LIN {X 0,Y 370.499,Z 396.613,A -85,B 0,C 180,E1 -12676.286,E2 -12676.286} C_VEL
LIN {X 0,Y 370.097,Z 408.814,A -85,B 0,C 180,E1 -12676.83,E2 -12676.83} C_VEL
LIN {X 0,Y 369.553,Z 419.294,A -85,B 0,C 180,E1 -12677.509,E2 -12677.509} C_VEL
LIN {X 0,Y 369.157,Z 427.534,A -85,B 0,C 180,E1 -12678.193,E2 -12678.193} C_VEL
LIN {X 0,Y 368.756,Z 436.851,A -85,B 0,C 180,E1 -12679.154,E2 -12679.154} C_VEL
LIN {X 0,Y 368.3,Z 446.273,A -85,B 0,C 180,E1 -12680.39,E2 -12680.39} C_VEL
LIN {X 0,Y 368.015,Z 452.98,A -85,B 0,C 180,E1 -12681.491,E2 -12681.491} C_VEL
LIN {X 0,Y 367.806,Z 458.55,A -85,B 0,C 180,E1 -12682.591,E2 -12682.591} C_VEL
LIN {X 0,Y 367.616,Z 463.595,A -85,B 0,C 180,E1 -12683.807,E2 -12683.807} C_VEL
LIN {X 0,Y 367.587,Z 467.801,A -85,B 0,C 180,E1 -12685.066,E2 -12685.066} C_VEL
LIN {X 0,Y 367.464,Z 470.726,A -85,B 0,C 180,E1 -12686.164,E2 -12686.164} C_VEL
LIN {X 0,Y 367.501,Z 473.873,A -85,B 0,C 180,E1 -12687.81,E2 -12687.81} C_VEL
LIN {X 0,Y 367.55,Z 475.255,A -85,B 0,C 180,E1 -12688.906,E2 -12688.906} C_VEL
LIN {X 0,Y 367.528,Z 476.096,A -85,B 0,C 180,E1 -12690.002,E2 -12690.002} C_VEL
LIN {X 0,Y 367.446,Z 476.353,A -85,B 0,C 180,E1 -12691.098,E2 -12691.098} C_VEL
LIN {X 0,Y 367.379,Z 475.995,A -85,B 0,C 180,E1 -12692.195,E2 -12692.195} C_VEL
LIN {X 0,Y 367.4,Z 475.12,A -85,B 0,C 180,E1 -12693.292,E2 -12693.292} C_VEL
LIN {X 0,Y 367.518,Z 473.725,A -85,B 0,C 180,E1 -12694.389,E2 -12694.389} C_VEL
LIN {X 0,Y 367.552,Z 471.788,A -85,B 0,C 180,E1 -12695.488,E2 -12695.488} C_VEL
LIN {X 0,Y 367.703,Z 469.247,A -85,B 0,C 180,E1 -12696.587,E2 -12696.587} C_VEL
LIN {X 0,Y 368.146,Z 464.102,A -85,B 0,C 180,E1 -12698.233,E2 -12698.233} C_VEL
LIN {X 0,Y 368.658,Z 458.565,A -85,B 0,C 180,E1 -12699.604,E2 -12699.604} C_VEL
LIN {X 0,Y 369.267,Z 453.206,A -85,B 0,C 180,E1 -12700.696,E2 -12700.696} C_VEL
LIN {X 0,Y 369.939,Z 446.802,A -85,B 0,C 180,E1 -12701.786,E2 -12701.786} C_VEL
LIN {X 0,Y 370.677,Z 439.081,A -85,B 0,C 180,E1 -12702.874,E2 -12702.874} C_VEL
LIN {X 0,Y 371.679,Z 429.594,A -85,B 0,C 180,E1 -12703.952,E2 -12703.952} C_VEL
LIN {X 0,Y 372.685,Z 418.758,A -85,B 0,C 180,E1 -12704.89,E2 -12704.89} C_VEL
LIN {X 0,Y 373.447,Z 409.895,A -85,B 0,C 180,E1 -12705.487,E2 -12705.487} C_VEL
LIN {X 0,Y 374.208,Z 399.587,A -85,B 0,C 180,E1 -12706.014,E2 -12706.014} C_VEL
LIN {X 0,Y 374.95,Z 384.489,A -85,B 0,C 180,E1 -12706.523,E2 -12706.523} C_VEL
LIN {X 0,Y 376.379,Z 344.678,A -85,B 0,C 180,E1 -12707.661,E2 -12707.661} C_VEL
LIN {X 0,Y 374.795,Z 331.794,A -85,B 0,C 180,E1 -12708.21,E2 -12708.21} C_VEL
LIN {X 0,Y 371.759,Z 316.775,A -85,B 0,C 180,E1 -12708.987,E2 -12708.987} C_VEL
LIN {X 0,Y 370.823,Z 312.912,A -85,B 0,C 180,E1 -12709.212,E2 -12709.212} C_VEL
LIN {X 0,Y 371.941,Z 296.849,A -85,B 0,C 180,E1 -12712.792,E2 -12712.792} C_VEL
LIN {X 0,Y 372.152,Z 293.067,A -85,B 0,C 180,E1 -12713.661,E2 -12713.661} C_VEL
LIN {X 0,Y 370.264,Z 284.467,A -85,B 0,C 180,E1 -12715.887,E2 -12715.887} C_VEL
LIN {X 0,Y 368.901,Z 279.352,A -85,B 0,C 180,E1 -12717.287,E2 -12717.287} C_VEL
LIN {X 0,Y 368.905,Z 279.348,A -85,B 0,C 180,E1 -12720.981,E2 -12720.981} C_VEL
LIN {X 0,Y 368.887,Z 279.348,A -85,B 0,C 180,E1 -12724.987,E2 -12724.987} C_VEL
LIN {X 0,Y 368.888,Z 279.346,A -85,B 0,C 180,E1 -12728.632,E2 -12728.632} C_VEL
LIN {X 0,Y 368.871,Z 279.346,A -85,B 0,C 180,E1 -12732.003,E2 -12732.003} C_VEL
LIN {X 0,Y 368.866,Z 279.35,A -85,B 0,C 180,E1 -12735.169,E2 -12735.169} C_VEL
LIN {X 0,Y 368.874,Z 279.344,A -85,B 0,C 180,E1 -12738.172,E2 -12738.172} C_VEL
LIN {X 0,Y 368.894,Z 279.342,A -85,B 0,C 180,E1 -12741.364,E2 -12741.364} C_VEL
LIN {X 0,Y 368.949,Z 279.338,A -85,B 0,C 180,E1 -12745.143,E2 -12745.143} C_VEL
LIN {X 0,Y 368.931,Z 279.342,A -85,B 0,C 180,E1 -12749.042,E2 -12749.042} C_VEL
LIN {X 0,Y 368.93,Z 279.345,A -85,B 0,C 180,E1 -12751.555,E2 -12751.555} C_VEL
LIN {X 0,Y 368.943,Z 279.346,A -85,B 0,C 180,E1 -12755.219,E2 -12755.219} C_VEL
LIN {X 0,Y 368.959,Z 279.518,A -85,B 0,C 180,E1 -12758.558,E2 -12758.558} C_VEL
LIN {X 0,Y 372.025,Z 289.625,A -85,B 0,C 180,E1 -12760.867,E2 -12760.867} C_VEL
LIN {X 0,Y 375.275,Z 296.975,A -85,B 0,C 180,E1 -12761.431,E2 -12761.431} C_VEL
LIN {X 0,Y 377.46,Z 310.343,A -85,B 0,C 180,E1 -12762.076,E2 -12762.076} C_VEL
LIN {X 0,Y 374.942,Z 371.825,A -85,B 0,C 180,E1 -12763.875,E2 -12763.875} C_VEL
LIN {X 0,Y 374.226,Z 384.155,A -85,B 0,C 180,E1 -12764.473,E2 -12764.473} C_VEL
LIN {X 0,Y 373.553,Z 393.994,A -85,B 0,C 180,E1 -12765.142,E2 -12765.142} C_VEL
LIN {X 0,Y 372.837,Z 403.308,A -85,B 0,C 180,E1 -12765.95,E2 -12765.95} C_VEL
LIN {X 0,Y 371.896,Z 413.125,A -85,B 0,C 180,E1 -12767.027,E2 -12767.027} C_VEL
LIN {X 0,Y 371.065,Z 421.69,A -85,B 0,C 180,E1 -12768.247,E2 -12768.247} C_VEL
LIN {X 0,Y 370.327,Z 427.955,A -85,B 0,C 180,E1 -12769.332,E2 -12769.332} C_VEL
LIN {X 0,Y 369.723,Z 433.161,A -85,B 0,C 180,E1 -12770.421,E2 -12770.421} C_VEL
LIN {X 0,Y 369.172,Z 437.83,A -85,B 0,C 180,E1 -12771.606,E2 -12771.606} C_VEL
LIN {X 0,Y 368.614,Z 442.264,A -85,B 0,C 180,E1 -12773.019,E2 -12773.019} C_VEL
LIN {X 0,Y 368.055,Z 445.796,A -85,B 0,C 180,E1 -12774.516,E2 -12774.516} C_VEL
LIN {X 0,Y 368.038,Z 447.581,A -85,B 0,C 180,E1 -12775.614,E2 -12775.614} C_VEL
LIN {X 0,Y 367.844,Z 448.849,A -85,B 0,C 180,E1 -12776.709,E2 -12776.709} C_VEL
LIN {X 0,Y 367.656,Z 449.603,A -85,B 0,C 180,E1 -12777.804,E2 -12777.804} C_VEL
LIN {X 0,Y 367.542,Z 449.826,A -85,B 0,C 180,E1 -12778.899,E2 -12778.899} C_VEL
LIN {X 0,Y 367.511,Z 449.429,A -85,B 0,C 180,E1 -12779.994,E2 -12779.994} C_VEL
LIN {X 0,Y 367.468,Z 448.484,A -85,B 0,C 180,E1 -12781.09,E2 -12781.09} C_VEL
LIN {X 0,Y 367.501,Z 446.123,A -85,B 0,C 180,E1 -12782.735,E2 -12782.735} C_VEL
LIN {X 0,Y 367.672,Z 442.383,A -85,B 0,C 180,E1 -12784.379,E2 -12784.379} C_VEL
LIN {X 0,Y 367.762,Z 437.898,A -85,B 0,C 180,E1 -12785.805,E2 -12785.805} C_VEL
LIN {X 0,Y 368.03,Z 432.871,A -85,B 0,C 180,E1 -12787.069,E2 -12787.069} C_VEL
LIN {X 0,Y 368.285,Z 427.255,A -85,B 0,C 180,E1 -12788.223,E2 -12788.223} C_VEL
LIN {X 0,Y 368.583,Z 420.783,A -85,B 0,C 180,E1 -12789.321,E2 -12789.321} C_VEL
LIN {X 0,Y 368.992,Z 412.939,A -85,B 0,C 180,E1 -12790.418,E2 -12790.418} C_VEL
LIN {X 0,Y 369.466,Z 403.205,A -85,B 0,C 180,E1 -12791.515,E2 -12791.515} C_VEL
LIN {X 0,Y 369.805,Z 393.743,A -85,B 0,C 180,E1 -12792.339,E2 -12792.339} C_VEL
LIN {X 0,Y 370.227,Z 383.654,A -85,B 0,C 180,E1 -12793.021,E2 -12793.021} C_VEL
LIN {X 0,Y 370.49,Z 372.702,A -85,B 0,C 180,E1 -12793.57,E2 -12793.57} C_VEL
LIN {X 0,Y 370.845,Z 357.09,A -85,B 0,C 180,E1 -12794.046,E2 -12794.046} C_VEL
LIN {X 0,Y 371.507,Z 307.956,A -85,B 0,C 180,E1 -12795.308,E2 -12795.308} C_VEL
LIN {X 0,Y 369.041,Z 290.368,A -85,B 0,C 180,E1 -12795.846,E2 -12795.846} C_VEL
LIN {X 0,Y 369.301,Z 282.159,A -85,B 0,C 180,E1 -12798.321,E2 -12798.321} C_VEL
LIN {X 0,Y 369.042,Z 279.327,A -85,B 0,C 180,E1 -12799.243,E2 -12799.243} C_VEL
LIN {X 0,Y 368.932,Z 279.341,A -85,B 0,C 180,E1 -12803.573,E2 -12803.573} C_VEL
LIN {X 0,Y 368.843,Z 279.351,A -85,B 0,C 180,E1 -12807.205,E2 -12807.205} C_VEL
LIN {X 0,Y 368.875,Z 279.347,A -85,B 0,C 180,E1 -12809.686,E2 -12809.686} C_VEL
LIN {X 0,Y 368.877,Z 279.347,A -85,B 0,C 180,E1 -12813.036,E2 -12813.036} C_VEL
LIN {X 0,Y 368.893,Z 279.348,A -85,B 0,C 180,E1 -12816.19,E2 -12816.19} C_VEL
LIN {X 0,Y 368.849,Z 279.353,A -85,B 0,C 180,E1 -12818.95,E2 -12818.95} C_VEL
LIN {X 0,Y 368.844,Z 279.351,A -85,B 0,C 180,E1 -12822.001,E2 -12822.001} C_VEL
LIN {X 0,Y 368.848,Z 279.352,A -85,B 0,C 180,E1 -12825.169,E2 -12825.169} C_VEL
LIN {X 0,Y 368.849,Z 279.351,A -85,B 0,C 180,E1 -12828.171,E2 -12828.171} C_VEL
LIN {X 0,Y 368.868,Z 279.35,A -85,B 0,C 180,E1 -12831.355,E2 -12831.355} C_VEL
LIN {X 0,Y 368.897,Z 279.347,A -85,B 0,C 180,E1 -12835.141,E2 -12835.141} C_VEL
LIN {X 0,Y 368.871,Z 279.35,A -85,B 0,C 180,E1 -12839.039,E2 -12839.039} C_VEL
LIN {X 0,Y 368.918,Z 279.343,A -85,B 0,C 180,E1 -12842.791,E2 -12842.791} C_VEL
LIN {X 0,Y 368.898,Z 279.344,A -85,B 0,C 180,E1 -12846.109,E2 -12846.109} C_VEL
LIN {X 0,Y 368.881,Z 279.348,A -85,B 0,C 180,E1 -12849.942,E2 -12849.942} C_VEL
LIN {X 0,Y 368.925,Z 279.344,A -85,B 0,C 180,E1 -12853.395,E2 -12853.395} C_VEL
LIN {X 0,Y 369.008,Z 279.33,A -85,B 0,C 180,E1 -12856.787,E2 -12856.787} C_VEL
LIN {X 0,Y 369.019,Z 279.331,A -85,B 0,C 180,E1 -12860.129,E2 -12860.129} C_VEL
LIN {X 0,Y 369.11,Z 279.319,A -85,B 0,C 180,E1 -12862.339,E2 -12862.339} C_VEL
LIN {X 0,Y 369.094,Z 279.32,A -85,B 0,C 180,E1 -12864.535,E2 -12864.535} C_VEL
LIN {X 0,Y 369.269,Z 279.301,A -85,B 0,C 180,E1 -12867.817,E2 -12867.817} C_VEL
LIN {X 0,Y 369.404,Z 279.284,A -85,B 0,C 180,E1 -12869.998,E2 -12869.998} C_VEL
LIN {X 0,Y 369.267,Z 279.301,A -85,B 0,C 180,E1 -12872.18,E2 -12872.18} C_VEL
LIN {X 0,Y 369.145,Z 279.316,A -85,B 0,C 180,E1 -12876.557,E2 -12876.557} C_VEL
LIN {X 0,Y 369.066,Z 279.324,A -85,B 0,C 180,E1 -12878.761,E2 -12878.761} C_VEL
LIN {X 0,Y 368.957,Z 279.34,A -85,B 0,C 180,E1 -12882.093,E2 -12882.093} C_VEL
LIN {X 0,Y 368.94,Z 279.338,A -85,B 0,C 180,E1 -12885.465,E2 -12885.465} C_VEL
LIN {X 0,Y 368.9,Z 279.346,A -85,B 0,C 180,E1 -12888.895,E2 -12888.895} C_VEL
LIN {X 0,Y 368.875,Z 279.35,A -85,B 0,C 180,E1 -12892.396,E2 -12892.396} C_VEL
LIN {X 0,Y 368.944,Z 279.338,A -85,B 0,C 180,E1 -12895.982,E2 -12895.982} C_VEL
LIN {X 0,Y 368.913,Z 279.345,A -85,B 0,C 180,E1 -12898.815,E2 -12898.815} C_VEL
LIN {X 0,Y 368.836,Z 279.351,A -85,B 0,C 180,E1 -12902.043,E2 -12902.043} C_VEL
LIN {X 0,Y 368.19,Z 279.435,A -85,B 0,C 180,E1 -12902.955,E2 -12902.955} C_VEL
LIN {X 0,Y 365.315,Z 279.791,A -85,B 0,C 180,E1 -12904.437,E2 -12904.437} C_VEL
LIN {X 0,Y 362.886,Z 280.093,A -85,B 0,C 180,E1 -12905.636,E2 -12905.636} C_VEL
LIN {X 0,Y 361.873,Z 280.221,A -85,B 0,C 180,E1 -12906.564,E2 -12906.564} C_VEL
LIN {X 0,Y 361.808,Z 280.229,A -85,B 0,C 180,E1 -12906.878,E2 -12906.878} C_VEL
LIN {X 0,Y 361.857,Z 280.223,A -85,B 0,C 180,E1 -12910.772,E2 -12910.772} C_VEL
LIN {X 0,Y 361.886,Z 280.217,A -85,B 0,C 180,E1 -12914.354,E2 -12914.354} C_VEL
LIN {X 0,Y 361.841,Z 280.227,A -85,B 0,C 180,E1 -12917.563,E2 -12917.563} C_VEL
LIN {X 0,Y 361.831,Z 280.226,A -85,B 0,C 180,E1 -12920.977,E2 -12920.977} C_VEL
LIN {X 0,Y 361.834,Z 280.223,A -85,B 0,C 180,E1 -12924.66,E2 -12924.66} C_VEL
LIN {X 0,Y 361.799,Z 280.228,A -85,B 0,C 180,E1 -12928.375,E2 -12928.375} C_VEL
LIN {X 0,Y 361.872,Z 280.22,A -85,B 0,C 180,E1 -12932.226,E2 -12932.226} C_VEL
LIN {X 0,Y 361.891,Z 280.216,A -85,B 0,C 180,E1 -12934.715,E2 -12934.715} C_VEL
LIN {X 0,Y 361.829,Z 280.226,A -85,B 0,C 180,E1 -12938.35,E2 -12938.35} C_VEL
LIN {X 0,Y 361.891,Z 280.22,A -85,B 0,C 180,E1 -12942.09,E2 -12942.09} C_VEL
LIN {X 0,Y 361.935,Z 280.211,A -85,B 0,C 180,E1 -12945.385,E2 -12945.385} C_VEL
LIN {X 0,Y 361.945,Z 280.21,A -85,B 0,C 180,E1 -12948.81,E2 -12948.81} C_VEL
LIN {X 0,Y 362.072,Z 280.197,A -85,B 0,C 180,E1 -12952.197,E2 -12952.197} C_VEL
LIN {X 0,Y 362.085,Z 280.196,A -85,B 0,C 180,E1 -12954.437,E2 -12954.437} C_VEL
LIN {X 0,Y 362.248,Z 280.173,A -85,B 0,C 180,E1 -12957.782,E2 -12957.782} C_VEL
LIN {X 0,Y 362.159,Z 280.184,A -85,B 0,C 180,E1 -12961.117,E2 -12961.117} C_VEL
LIN {X 0,Y 362.256,Z 280.174,A -85,B 0,C 180,E1 -12962.229,E2 -12962.229} C_VEL
LIN {X 0,Y 362.11,Z 280.193,A -85,B 0,C 180,E1 -12966.693,E2 -12966.693} C_VEL
LIN {X 0,Y 361.988,Z 280.205,A -85,B 0,C 180,E1 -12970.068,E2 -12970.068} C_VEL
LIN {X 0,Y 361.97,Z 280.206,A -85,B 0,C 180,E1 -12973.892,E2 -12973.892} C_VEL
LIN {X 0,Y 361.88,Z 280.218,A -85,B 0,C 180,E1 -12978.108,E2 -12978.108} C_VEL
LIN {X 0,Y 361.848,Z 280.223,A -85,B 0,C 180,E1 -12981.66,E2 -12981.66} C_VEL
LIN {X 0,Y 361.857,Z 280.225,A -85,B 0,C 180,E1 -12985.3,E2 -12985.3} C_VEL
LIN {X 0,Y 361.853,Z 280.225,A -85,B 0,C 180,E1 -12989.078,E2 -12989.078} C_VEL
LIN {X 0,Y 361.846,Z 280.224,A -85,B 0,C 180,E1 -12992.95,E2 -12992.95} C_VEL
LIN {X 0,Y 361.862,Z 280.224,A -85,B 0,C 180,E1 -12995.642,E2 -12995.642} C_VEL
LIN {X 0,Y 361.825,Z 280.226,A -85,B 0,C 180,E1 -12999.022,E2 -12999.022} C_VEL
LIN {X 0,Y 361.83,Z 280.224,A -85,B 0,C 180,E1 -13002.834,E2 -13002.834} C_VEL
LIN {X 0,Y 361.814,Z 280.231,A -85,B 0,C 180,E1 -13005.952,E2 -13005.952} C_VEL
LIN {X 0,Y 361.813,Z 280.227,A -85,B 0,C 180,E1 -13009.254,E2 -13009.254} C_VEL
LIN {X 0,Y 361.865,Z 280.219,A -85,B 0,C 180,E1 -13012.985,E2 -13012.985} C_VEL
LIN {X 0,Y 361.863,Z 280.221,A -85,B 0,C 180,E1 -13016.635,E2 -13016.635} C_VEL
LIN {X 0,Y 361.853,Z 280.223,A -85,B 0,C 180,E1 -13019.673,E2 -13019.673} C_VEL
LIN {X 0,Y 361.968,Z 280.278,A -85,B 0,C 180,E1 -13024.099,E2 -13024.099} C_VEL
LIN {X 0,Y 363.512,Z 289.449,A -85,B 0,C 180,E1 -13026.653,E2 -13026.653} C_VEL
LIN {X 0,Y 363.468,Z 293.753,A -85,B 0,C 180,E1 -13027.801,E2 -13027.801} C_VEL
LIN {X 0,Y 362.434,Z 307.198,A -85,B 0,C 180,E1 -13031.342,E2 -13031.342} C_VEL
LIN {X 0,Y 361.788,Z 317.108,A -85,B 0,C 180,E1 -13033.932,E2 -13033.932} C_VEL
LIN {X 0,Y 364.043,Z 340.993,A -85,B 0,C 180,E1 -13034.665,E2 -13034.665} C_VEL
LIN {X 0,Y 364.324,Z 346.449,A -85,B 0,C 180,E1 -13034.82,E2 -13034.82} C_VEL
LIN {X 0,Y 363.447,Z 395.966,A -85,B 0,C 180,E1 -13036.157,E2 -13036.157} C_VEL
LIN {X 0,Y 363.049,Z 408.33,A -85,B 0,C 180,E1 -13036.712,E2 -13036.712} C_VEL
LIN {X 0,Y 362.494,Z 418.839,A -85,B 0,C 180,E1 -13037.404,E2 -13037.404} C_VEL
LIN {X 0,Y 362.204,Z 425.633,A -85,B 0,C 180,E1 -13037.963,E2 -13037.963} C_VEL
LIN {X 0,Y 361.736,Z 433.963,A -85,B 0,C 180,E1 -13038.799,E2 -13038.799} C_VEL
LIN {X 0,Y 361.441,Z 440.9,A -85,B 0,C 180,E1 -13039.64,E2 -13039.64} C_VEL
LIN {X 0,Y 361.168,Z 446.8,A -85,B 0,C 180,E1 -13040.481,E2 -13040.481} C_VEL
LIN {X 0,Y 360.903,Z 453.387,A -85,B 0,C 180,E1 -13041.604,E2 -13041.604} C_VEL
LIN {X 0,Y 360.712,Z 458.837,A -85,B 0,C 180,E1 -13042.726,E2 -13042.726} C_VEL
LIN {X 0,Y 360.549,Z 463.2,A -85,B 0,C 180,E1 -13043.804,E2 -13043.804} C_VEL
LIN {X 0,Y 360.497,Z 467.086,A -85,B 0,C 180,E1 -13044.969,E2 -13044.969} C_VEL
LIN {X 0,Y 360.397,Z 470.113,A -85,B 0,C 180,E1 -13046.088,E2 -13046.088} C_VEL
LIN {X 0,Y 360.406,Z 473.349,A -85,B 0,C 180,E1 -13047.767,E2 -13047.767} C_VEL
LIN {X 0,Y 360.467,Z 474.826,A -85,B 0,C 180,E1 -13048.885,E2 -13048.885} C_VEL
LIN {X 0,Y 360.464,Z 475.744,A -85,B 0,C 180,E1 -13050.002,E2 -13050.002} C_VEL
LIN {X 0,Y 360.35,Z 476.026,A -85,B 0,C 180,E1 -13051.119,E2 -13051.119} C_VEL
LIN {X 0,Y 360.283,Z 475.753,A -85,B 0,C 180,E1 -13052.238,E2 -13052.238} C_VEL
LIN {X 0,Y 360.322,Z 474.969,A -85,B 0,C 180,E1 -13053.356,E2 -13053.356} C_VEL
LIN {X 0,Y 360.427,Z 473.661,A -85,B 0,C 180,E1 -13054.475,E2 -13054.475} C_VEL
LIN {X 0,Y 360.47,Z 471.798,A -85,B 0,C 180,E1 -13055.596,E2 -13055.596} C_VEL
LIN {X 0,Y 360.79,Z 467.77,A -85,B 0,C 180,E1 -13057.276,E2 -13057.276} C_VEL
LIN {X 0,Y 361.326,Z 462.323,A -85,B 0,C 180,E1 -13058.954,E2 -13058.954} C_VEL
LIN {X 0,Y 362.012,Z 456.497,A -85,B 0,C 180,E1 -13060.347,E2 -13060.347} C_VEL
LIN {X 0,Y 362.869,Z 449.22,A -85,B 0,C 180,E1 -13061.735,E2 -13061.735} C_VEL
LIN {X 0,Y 363.717,Z 440.961,A -85,B 0,C 180,E1 -13062.983,E2 -13062.983} C_VEL
LIN {X 0,Y 364.608,Z 433.136,A -85,B 0,C 180,E1 -13063.944,E2 -13063.944} C_VEL
LIN {X 0,Y 365.438,Z 425.126,A -85,B 0,C 180,E1 -13064.765,E2 -13064.765} C_VEL
LIN {X 0,Y 366.408,Z 415.242,A -85,B 0,C 180,E1 -13065.579,E2 -13065.579} C_VEL
LIN {X 0,Y 367.489,Z 403.009,A -85,B 0,C 180,E1 -13066.315,E2 -13066.315} C_VEL
LIN {X 0,Y 368.205,Z 392.162,A -85,B 0,C 180,E1 -13066.762,E2 -13066.762} C_VEL
LIN {X 0,Y 370.064,Z 345.467,A -85,B 0,C 180,E1 -13068.146,E2 -13068.146} C_VEL
LIN {X 0,Y 368.584,Z 333.165,A -85,B 0,C 180,E1 -13068.705,E2 -13068.705} C_VEL
LIN {X 0,Y 365.594,Z 318.278,A -85,B 0,C 180,E1 -13069.513,E2 -13069.513} C_VEL
LIN {X 0,Y 364.175,Z 312.447,A -85,B 0,C 180,E1 -13069.865,E2 -13069.865} C_VEL
LIN {X 0,Y 365.305,Z 297.746,A -85,B 0,C 180,E1 -13073.23,E2 -13073.23} C_VEL
LIN {X 0,Y 365.277,Z 294.118,A -85,B 0,C 180,E1 -13074.092,E2 -13074.092} C_VEL
LIN {X 0,Y 363.265,Z 285.529,A -85,B 0,C 180,E1 -13076.423,E2 -13076.423} C_VEL
LIN {X 0,Y 361.884,Z 280.227,A -85,B 0,C 180,E1 -13077.979,E2 -13077.979} C_VEL
LIN {X 0,Y 361.82,Z 280.228,A -85,B 0,C 180,E1 -13081.633,E2 -13081.633} C_VEL
LIN {X 0,Y 361.85,Z 280.225,A -85,B 0,C 180,E1 -13085.334,E2 -13085.334} C_VEL
LIN {X 0,Y 361.839,Z 280.228,A -85,B 0,C 180,E1 -13089.016,E2 -13089.016} C_VEL
LIN {X 0,Y 361.824,Z 280.229,A -85,B 0,C 180,E1 -13092.832,E2 -13092.832} C_VEL
LIN {X 0,Y 361.802,Z 280.226,A -85,B 0,C 180,E1 -13095.951,E2 -13095.951} C_VEL
LIN {X 0,Y 361.828,Z 280.224,A -85,B 0,C 180,E1 -13099.248,E2 -13099.248} C_VEL
LIN {X 0,Y 361.88,Z 280.219,A -85,B 0,C 180,E1 -13102.979,E2 -13102.979} C_VEL
LIN {X 0,Y 361.876,Z 280.221,A -85,B 0,C 180,E1 -13106.629,E2 -13106.629} C_VEL
LIN {X 0,Y 361.874,Z 280.222,A -85,B 0,C 180,E1 -13109.667,E2 -13109.667} C_VEL
LIN {X 0,Y 361.881,Z 280.224,A -85,B 0,C 180,E1 -13113.465,E2 -13113.465} C_VEL
LIN {X 0,Y 361.894,Z 280.224,A -85,B 0,C 180,E1 -13117.14,E2 -13117.14} C_VEL
LIN {X 0,Y 361.94,Z 280.365,A -85,B 0,C 180,E1 -13117.821,E2 -13117.821} C_VEL
LIN {X 0,Y 364.984,Z 290.172,A -85,B 0,C 180,E1 -13120.18,E2 -13120.18} C_VEL
LIN {X 0,Y 369.442,Z 299.787,A -85,B 0,C 180,E1 -13120.978,E2 -13120.978} C_VEL
LIN {X 0,Y 371.267,Z 311.235,A -85,B 0,C 180,E1 -13121.557,E2 -13121.557} C_VEL
LIN {X 0,Y 368.557,Z 372.344,A -85,B 0,C 180,E1 -13123.41,E2 -13123.41} C_VEL
LIN {X 0,Y 367.841,Z 384.041,A -85,B 0,C 180,E1 -13123.983,E2 -13123.983} C_VEL
LIN {X 0,Y 367.166,Z 393.07,A -85,B 0,C 180,E1 -13124.594,E2 -13124.594} C_VEL
LIN {X 0,Y 366.368,Z 402.518,A -85,B 0,C 180,E1 -13125.413,E2 -13125.413} C_VEL
LIN {X 0,Y 365.343,Z 412.548,A -85,B 0,C 180,E1 -13126.507,E2 -13126.507} C_VEL
LIN {X 0,Y 364.423,Z 421.268,A -85,B 0,C 180,E1 -13127.747,E2 -13127.747} C_VEL
LIN {X 0,Y 363.598,Z 427.668,A -85,B 0,C 180,E1 -13128.85,E2 -13128.85} C_VEL
LIN {X 0,Y 362.793,Z 434.168,A -85,B 0,C 180,E1 -13130.236,E2 -13130.236} C_VEL
LIN {X 0,Y 362.217,Z 438.717,A -85,B 0,C 180,E1 -13131.444,E2 -13131.444} C_VEL
LIN {X 0,Y 361.597,Z 443.122,A -85,B 0,C 180,E1 -13132.917,E2 -13132.917} C_VEL
LIN {X 0,Y 361.014,Z 446.43,A -85,B 0,C 180,E1 -13134.409,E2 -13134.409} C_VEL
LIN {X 0,Y 360.98,Z 448.107,A -85,B 0,C 180,E1 -13135.528,E2 -13135.528} C_VEL
LIN {X 0,Y 360.767,Z 449.279,A -85,B 0,C 180,E1 -13136.644,E2 -13136.644} C_VEL
LIN {X 0,Y 360.569,Z 449.94,A -85,B 0,C 180,E1 -13137.76,E2 -13137.76} C_VEL
LIN {X 0,Y 360.449,Z 450.086,A -85,B 0,C 180,E1 -13138.877,E2 -13138.877} C_VEL
LIN {X 0,Y 360.414,Z 449.654,A -85,B 0,C 180,E1 -13139.994,E2 -13139.994} C_VEL
LIN {X 0,Y 360.37,Z 448.616,A -85,B 0,C 180,E1 -13141.112,E2 -13141.112} C_VEL
LIN {X 0,Y 360.41,Z 446.123,A -85,B 0,C 180,E1 -13142.788,E2 -13142.788} C_VEL
LIN {X 0,Y 360.605,Z 442.179,A -85,B 0,C 180,E1 -13144.465,E2 -13144.465} C_VEL
LIN {X 0,Y 360.688,Z 436.997,A -85,B 0,C 180,E1 -13146.077,E2 -13146.077} C_VEL
LIN {X 0,Y 360.982,Z 432.163,A -85,B 0,C 180,E1 -13147.264,E2 -13147.264} C_VEL
LIN {X 0,Y 361.232,Z 426.65,A -85,B 0,C 180,E1 -13148.384,E2 -13148.384} C_VEL
LIN {X 0,Y 361.663,Z 418.231,A -85,B 0,C 180,E1 -13149.784,E2 -13149.784} C_VEL
LIN {X 0,Y 362.053,Z 409.628,A -85,B 0,C 180,E1 -13150.903,E2 -13150.903} C_VEL
LIN {X 0,Y 362.449,Z 401.766,A -85,B 0,C 180,E1 -13151.741,E2 -13151.741} C_VEL
LIN {X 0,Y 362.858,Z 391.964,A -85,B 0,C 180,E1 -13152.579,E2 -13152.579} C_VEL
LIN {X 0,Y 363.292,Z 381.401,A -85,B 0,C 180,E1 -13153.274,E2 -13153.274} C_VEL
LIN {X 0,Y 363.518,Z 368.943,A -85,B 0,C 180,E1 -13153.836,E2 -13153.836} C_VEL
LIN {X 0,Y 364.566,Z 309.148,A -85,B 0,C 180,E1 -13155.441,E2 -13155.441} C_VEL
LIN {X 0,Y 361.992,Z 290.643,A -85,B 0,C 180,E1 -13156.018,E2 -13156.018} C_VEL
LIN {X 0,Y 362.284,Z 283.853,A -85,B 0,C 180,E1 -13158.089,E2 -13158.089} C_VEL
LIN {X 0,Y 362.015,Z 280.202,A -85,B 0,C 180,E1 -13159.264,E2 -13159.264} C_VEL
LIN {X 0,Y 361.863,Z 280.22,A -85,B 0,C 180,E1 -13162.85,E2 -13162.85} C_VEL
LIN {X 0,Y 361.841,Z 280.226,A -85,B 0,C 180,E1 -13166.526,E2 -13166.526} C_VEL
LIN {X 0,Y 361.829,Z 280.228,A -85,B 0,C 180,E1 -13170.324,E2 -13170.324} C_VEL
LIN {X 0,Y 361.833,Z 280.227,A -85,B 0,C 180,E1 -13174.274,E2 -13174.274} C_VEL
LIN {X 0,Y 361.836,Z 280.224,A -85,B 0,C 180,E1 -13177.215,E2 -13177.215} C_VEL
LIN {X 0,Y 361.786,Z 280.233,A -85,B 0,C 180,E1 -13180.744,E2 -13180.744} C_VEL
LIN {X 0,Y 361.786,Z 280.232,A -85,B 0,C 180,E1 -13184.362,E2 -13184.362} C_VEL
LIN {X 0,Y 361.803,Z 280.228,A -85,B 0,C 180,E1 -13187.562,E2 -13187.562} C_VEL
LIN {X 0,Y 361.83,Z 280.228,A -85,B 0,C 180,E1 -13190.968,E2 -13190.968} C_VEL
LIN {X 0,Y 361.836,Z 280.226,A -85,B 0,C 180,E1 -13194.65,E2 -13194.65} C_VEL
LIN {X 0,Y 361.796,Z 280.228,A -85,B 0,C 180,E1 -13198.365,E2 -13198.365} C_VEL
LIN {X 0,Y 361.864,Z 280.22,A -85,B 0,C 180,E1 -13202.216,E2 -13202.216} C_VEL
LIN {X 0,Y 361.883,Z 280.218,A -85,B 0,C 180,E1 -13204.705,E2 -13204.705} C_VEL
LIN {X 0,Y 361.836,Z 280.223,A -85,B 0,C 180,E1 -13208.342,E2 -13208.342} C_VEL
LIN {X 0,Y 361.919,Z 280.214,A -85,B 0,C 180,E1 -13212.057,E2 -13212.057} C_VEL
LIN {X 0,Y 361.947,Z 280.211,A -85,B 0,C 180,E1 -13216.098,E2 -13216.098} C_VEL
LIN {X 0,Y 361.983,Z 280.209,A -85,B 0,C 180,E1 -13219.935,E2 -13219.935} C_VEL
LIN {X 0,Y 362.113,Z 280.19,A -85,B 0,C 180,E1 -13223.311,E2 -13223.311} C_VEL
LIN {X 0,Y 362.234,Z 280.177,A -85,B 0,C 180,E1 -13227.774,E2 -13227.774} C_VEL
LIN {X 0,Y 362.374,Z 280.16,A -85,B 0,C 180,E1 -13229.998,E2 -13229.998} C_VEL
LIN {X 0,Y 362.233,Z 280.178,A -85,B 0,C 180,E1 -13232.222,E2 -13232.222} C_VEL
LIN {X 0,Y 362.107,Z 280.191,A -85,B 0,C 180,E1 -13236.685,E2 -13236.685} C_VEL
LIN {X 0,Y 361.98,Z 280.209,A -85,B 0,C 180,E1 -13240.061,E2 -13240.061} C_VEL
LIN {X 0,Y 361.942,Z 280.212,A -85,B 0,C 180,E1 -13243.899,E2 -13243.899} C_VEL
LIN {X 0,Y 361.911,Z 280.215,A -85,B 0,C 180,E1 -13247.939,E2 -13247.939} C_VEL
LIN {X 0,Y 361.827,Z 280.224,A -85,B 0,C 180,E1 -13251.655,E2 -13251.655} C_VEL
LIN {X 0,Y 361.873,Z 280.22,A -85,B 0,C 180,E1 -13255.292,E2 -13255.292} C_VEL
LIN {X 0,Y 361.868,Z 280.219,A -85,B 0,C 180,E1 -13257.78,E2 -13257.78} C_VEL
LIN {X 0,Y 361.794,Z 280.231,A -85,B 0,C 180,E1 -13261.287,E2 -13261.287} C_VEL
LIN {X 0,Y 361.802,Z 280.228,A -85,B 0,C 180,E1 -13264.283,E2 -13264.283} C_VEL
LIN {X 0,Y 361.808,Z 280.229,A -85,B 0,C 180,E1 -13266.878,E2 -13266.878} C_VEL
LIN {X 0,Y 361.184,Z 280.313,A -85,B 0,C 180,E1 -13267.807,E2 -13267.807} C_VEL
LIN {X 0,Y 358.334,Z 280.67,A -85,B 0,C 180,E1 -13269.316,E2 -13269.316} C_VEL
LIN {X 0,Y 355.896,Z 280.968,A -85,B 0,C 180,E1 -13270.538,E2 -13270.538} C_VEL
LIN {X 0,Y 354.854,Z 281.096,A -85,B 0,C 180,E1 -13271.483,E2 -13271.483} C_VEL
LIN {X 0,Y 354.773,Z 281.103,A -85,B 0,C 180,E1 -13271.803,E2 -13271.803} C_VEL
LIN {X 0,Y 354.841,Z 281.099,A -85,B 0,C 180,E1 -13275.477,E2 -13275.477} C_VEL
LIN {X 0,Y 354.812,Z 281.102,A -85,B 0,C 180,E1 -13279.193,E2 -13279.193} C_VEL
LIN {X 0,Y 354.767,Z 281.103,A -85,B 0,C 180,E1 -13282.407,E2 -13282.407} C_VEL
LIN {X 0,Y 354.771,Z 281.104,A -85,B 0,C 180,E1 -13284.945,E2 -13284.945} C_VEL
LIN {X 0,Y 354.755,Z 281.105,A -85,B 0,C 180,E1 -13288.41,E2 -13288.41} C_VEL
LIN {X 0,Y 354.81,Z 281.102,A -85,B 0,C 180,E1 -13291.624,E2 -13291.624} C_VEL
LIN {X 0,Y 354.863,Z 281.094,A -85,B 0,C 180,E1 -13294.178,E2 -13294.178} C_VEL
LIN {X 0,Y 354.783,Z 281.106,A -85,B 0,C 180,E1 -13297.898,E2 -13297.898} C_VEL
LIN {X 0,Y 354.861,Z 281.096,A -85,B 0,C 180,E1 -13301.914,E2 -13301.914} C_VEL
LIN {X 0,Y 354.917,Z 281.089,A -85,B 0,C 180,E1 -13305.987,E2 -13305.987} C_VEL
LIN {X 0,Y 354.932,Z 281.085,A -85,B 0,C 180,E1 -13309.741,E2 -13309.741} C_VEL
LIN {X 0,Y 355.088,Z 281.063,A -85,B 0,C 180,E1 -13313.186,E2 -13313.186} C_VEL
LIN {X 0,Y 355.211,Z 281.049,A -85,B 0,C 180,E1 -13317.738,E2 -13317.738} C_VEL
LIN {X 0,Y 355.13,Z 281.059,A -85,B 0,C 180,E1 -13321.14,E2 -13321.14} C_VEL
LIN {X 0,Y 355.218,Z 281.051,A -85,B 0,C 180,E1 -13322.273,E2 -13322.273} C_VEL
LIN {X 0,Y 355.075,Z 281.07,A -85,B 0,C 180,E1 -13326.826,E2 -13326.826} C_VEL
LIN {X 0,Y 354.944,Z 281.083,A -85,B 0,C 180,E1 -13330.27,E2 -13330.27} C_VEL
LIN {X 0,Y 354.914,Z 281.085,A -85,B 0,C 180,E1 -13334.011,E2 -13334.011} C_VEL
LIN {X 0,Y 354.838,Z 281.095,A -85,B 0,C 180,E1 -13338.075,E2 -13338.075} C_VEL
LIN {X 0,Y 354.801,Z 281.099,A -85,B 0,C 180,E1 -13342.113,E2 -13342.113} C_VEL
LIN {X 0,Y 354.8,Z 281.1,A -85,B 0,C 180,E1 -13345.84,E2 -13345.84} C_VEL
LIN {X 0,Y 354.794,Z 281.103,A -85,B 0,C 180,E1 -13349.689,E2 -13349.689} C_VEL
LIN {X 0,Y 354.785,Z 281.101,A -85,B 0,C 180,E1 -13352.338,E2 -13352.338} C_VEL
LIN {X 0,Y 354.817,Z 281.102,A -85,B 0,C 180,E1 -13355.703,E2 -13355.703} C_VEL
LIN {X 0,Y 354.77,Z 281.107,A -85,B 0,C 180,E1 -13359.417,E2 -13359.417} C_VEL
LIN {X 0,Y 354.782,Z 281.102,A -85,B 0,C 180,E1 -13362.87,E2 -13362.87} C_VEL
LIN {X 0,Y 354.764,Z 281.107,A -85,B 0,C 180,E1 -13366.107,E2 -13366.107} C_VEL
LIN {X 0,Y 354.766,Z 281.104,A -85,B 0,C 180,E1 -13369.179,E2 -13369.179} C_VEL
LIN {X 0,Y 354.803,Z 281.101,A -85,B 0,C 180,E1 -13372.409,E2 -13372.409} C_VEL
LIN {X 0,Y 354.812,Z 281.098,A -85,B 0,C 180,E1 -13374.944,E2 -13374.944} C_VEL
LIN {X 0,Y 354.799,Z 281.103,A -85,B 0,C 180,E1 -13378.409,E2 -13378.409} C_VEL
LIN {X 0,Y 354.797,Z 281.101,A -85,B 0,C 180,E1 -13381.617,E2 -13381.617} C_VEL
LIN {X 0,Y 354.927,Z 281.165,A -85,B 0,C 180,E1 -13384.02,E2 -13384.02} C_VEL
LIN {X 0,Y 356.521,Z 290.93,A -85,B 0,C 180,E1 -13386.783,E2 -13386.783} C_VEL
LIN {X 0,Y 356.146,Z 297.616,A -85,B 0,C 180,E1 -13388.591,E2 -13388.591} C_VEL
LIN {X 0,Y 355.098,Z 311.221,A -85,B 0,C 180,E1 -13392.239,E2 -13392.239} C_VEL
LIN {X 0,Y 354.747,Z 316.873,A -85,B 0,C 180,E1 -13393.752,E2 -13393.752} C_VEL
LIN {X 0,Y 356.836,Z 340.224,A -85,B 0,C 180,E1 -13394.481,E2 -13394.481} C_VEL
LIN {X 0,Y 357.3,Z 346.445,A -85,B 0,C 180,E1 -13394.666,E2 -13394.666} C_VEL
LIN {X 0,Y 356.392,Z 396.06,A -85,B 0,C 180,E1 -13396.059,E2 -13396.059} C_VEL
LIN {X 0,Y 355.982,Z 408.764,A -85,B 0,C 180,E1 -13396.661,E2 -13396.661} C_VEL
LIN {X 0,Y 355.468,Z 418.171,A -85,B 0,C 180,E1 -13397.296,E2 -13397.296} C_VEL
LIN {X 0,Y 355.058,Z 426.492,A -85,B 0,C 180,E1 -13398.007,E2 -13398.007} C_VEL
LIN {X 0,Y 354.612,Z 434.614,A -85,B 0,C 180,E1 -13398.861,E2 -13398.861} C_VEL
LIN {X 0,Y 354.326,Z 441.392,A -85,B 0,C 180,E1 -13399.719,E2 -13399.719} C_VEL
LIN {X 0,Y 353.992,Z 448.916,A -85,B 0,C 180,E1 -13400.863,E2 -13400.863} C_VEL
LIN {X 0,Y 353.687,Z 456.541,A -85,B 0,C 180,E1 -13402.294,E2 -13402.294} C_VEL
LIN {X 0,Y 353.486,Z 462.699,A -85,B 0,C 180,E1 -13403.795,E2 -13403.795} C_VEL
LIN {X 0,Y 353.42,Z 467.898,A -85,B 0,C 180,E1 -13405.44,E2 -13405.44} C_VEL
LIN {X 0,Y 353.27,Z 470.655,A -85,B 0,C 180,E1 -13406.58,E2 -13406.58} C_VEL
LIN {X 0,Y 353.312,Z 472.811,A -85,B 0,C 180,E1 -13407.722,E2 -13407.722} C_VEL
LIN {X 0,Y 353.387,Z 474.391,A -85,B 0,C 180,E1 -13408.862,E2 -13408.862} C_VEL
LIN {X 0,Y 353.4,Z 475.351,A -85,B 0,C 180,E1 -13410.002,E2 -13410.002} C_VEL
LIN {X 0,Y 353.254,Z 475.691,A -85,B 0,C 180,E1 -13411.142,E2 -13411.142} C_VEL
LIN {X 0,Y 353.191,Z 475.511,A -85,B 0,C 180,E1 -13412.283,E2 -13412.283} C_VEL
LIN {X 0,Y 353.246,Z 474.82,A -85,B 0,C 180,E1 -13413.424,E2 -13413.424} C_VEL
LIN {X 0,Y 353.34,Z 473.614,A -85,B 0,C 180,E1 -13414.565,E2 -13414.565} C_VEL
LIN {X 0,Y 353.421,Z 471.007,A -85,B 0,C 180,E1 -13416.108,E2 -13416.108} C_VEL
LIN {X 0,Y 353.74,Z 467.958,A -85,B 0,C 180,E1 -13417.422,E2 -13417.422} C_VEL
LIN {X 0,Y 354.185,Z 463.634,A -85,B 0,C 180,E1 -13418.848,E2 -13418.848} C_VEL
LIN {X 0,Y 354.858,Z 458.145,A -85,B 0,C 180,E1 -13420.269,E2 -13420.269} C_VEL
LIN {X 0,Y 355.764,Z 451.326,A -85,B 0,C 180,E1 -13421.684,E2 -13421.684} C_VEL
LIN {X 0,Y 356.81,Z 442.933,A -85,B 0,C 180,E1 -13423.094,E2 -13423.094} C_VEL
LIN {X 0,Y 357.804,Z 434.433,A -85,B 0,C 180,E1 -13424.215,E2 -13424.215} C_VEL
LIN {X 0,Y 358.864,Z 425.266,A -85,B 0,C 180,E1 -13425.187,E2 -13425.187} C_VEL
LIN {X 0,Y 359.875,Z 415.474,A -85,B 0,C 180,E1 -13426.014,E2 -13426.014} C_VEL
LIN {X 0,Y 361.086,Z 402.868,A -85,B 0,C 180,E1 -13426.795,E2 -13426.795} C_VEL
LIN {X 0,Y 361.833,Z 392.185,A -85,B 0,C 180,E1 -13427.248,E2 -13427.248} C_VEL
LIN {X 0,Y 363.831,Z 346.023,A -85,B 0,C 180,E1 -13428.685,E2 -13428.685} C_VEL
LIN {X 0,Y 362.177,Z 333.049,A -85,B 0,C 180,E1 -13429.304,E2 -13429.304} C_VEL
LIN {X 0,Y 359.236,Z 318.599,A -85,B 0,C 180,E1 -13430.146,E2 -13430.146} C_VEL
LIN {X 0,Y 357.604,Z 311.842,A -85,B 0,C 180,E1 -13430.607,E2 -13430.607} C_VEL
LIN {X 0,Y 358.718,Z 298.733,A -85,B 0,C 180,E1 -13433.682,E2 -13433.682} C_VEL
LIN {X 0,Y 358.638,Z 296.277,A -85,B 0,C 180,E1 -13434.302,E2 -13434.302} C_VEL
LIN {X 0,Y 356.694,Z 287.997,A -85,B 0,C 180,E1 -13436.633,E2 -13436.633} C_VEL
LIN {X 0,Y 354.845,Z 281.103,A -85,B 0,C 180,E1 -13438.722,E2 -13438.722} C_VEL
LIN {X 0,Y 354.768,Z 281.107,A -85,B 0,C 180,E1 -13442.337,E2 -13442.337} C_VEL
LIN {X 0,Y 354.805,Z 281.102,A -85,B 0,C 180,E1 -13445.69,E2 -13445.69} C_VEL
LIN {X 0,Y 354.788,Z 281.102,A -85,B 0,C 180,E1 -13449.412,E2 -13449.412} C_VEL
LIN {X 0,Y 354.779,Z 281.107,A -85,B 0,C 180,E1 -13452.861,E2 -13452.861} C_VEL
LIN {X 0,Y 354.755,Z 281.104,A -85,B 0,C 180,E1 -13456.097,E2 -13456.097} C_VEL
LIN {X 0,Y 354.78,Z 281.102,A -85,B 0,C 180,E1 -13459.173,E2 -13459.173} C_VEL
LIN {X 0,Y 354.817,Z 281.095,A -85,B 0,C 180,E1 -13462.403,E2 -13462.403} C_VEL
LIN {X 0,Y 354.827,Z 281.099,A -85,B 0,C 180,E1 -13464.938,E2 -13464.938} C_VEL
LIN {X 0,Y 354.812,Z 281.102,A -85,B 0,C 180,E1 -13468.403,E2 -13468.403} C_VEL
LIN {X 0,Y 354.818,Z 281.103,A -85,B 0,C 180,E1 -13471.611,E2 -13471.611} C_VEL
LIN {X 0,Y 354.852,Z 281.103,A -85,B 0,C 180,E1 -13475.654,E2 -13475.654} C_VEL
LIN {X 0,Y 354.846,Z 281.134,A -85,B 0,C 180,E1 -13476.968,E2 -13476.968} C_VEL
LIN {X 0,Y 357.982,Z 290.845,A -85,B 0,C 180,E1 -13479.438,E2 -13479.438} C_VEL
LIN {X 0,Y 363.598,Z 302.528,A -85,B 0,C 180,E1 -13480.5,E2 -13480.5} C_VEL
LIN {X 0,Y 365.137,Z 312.378,A -85,B 0,C 180,E1 -13481.018,E2 -13481.018} C_VEL
LIN {X 0,Y 362.246,Z 372.23,A -85,B 0,C 180,E1 -13482.895,E2 -13482.895} C_VEL
LIN {X 0,Y 361.485,Z 383.971,A -85,B 0,C 180,E1 -13483.476,E2 -13483.476} C_VEL
LIN {X 0,Y 360.676,Z 393.91,A -85,B 0,C 180,E1 -13484.164,E2 -13484.164} C_VEL
LIN {X 0,Y 359.82,Z 403.279,A -85,B 0,C 180,E1 -13484.996,E2 -13484.996} C_VEL
LIN {X 0,Y 358.74,Z 413.222,A -85,B 0,C 180,E1 -13486.109,E2 -13486.109} C_VEL
LIN {X 0,Y 357.859,Z 421.012,A -85,B 0,C 180,E1 -13487.231,E2 -13487.231} C_VEL
LIN {X 0,Y 356.986,Z 427.462,A -85,B 0,C 180,E1 -13488.353,E2 -13488.353} C_VEL
LIN {X 0,Y 356.204,Z 432.844,A -85,B 0,C 180,E1 -13489.479,E2 -13489.479} C_VEL
LIN {X 0,Y 355.67,Z 436.348,A -85,B 0,C 180,E1 -13490.326,E2 -13490.326} C_VEL
LIN {X 0,Y 354.965,Z 441.864,A -85,B 0,C 180,E1 -13492.028,E2 -13492.028} C_VEL
LIN {X 0,Y 354.146,Z 445.945,A -85,B 0,C 180,E1 -13493.728,E2 -13493.728} C_VEL
LIN {X 0,Y 353.974,Z 447.061,A -85,B 0,C 180,E1 -13494.297,E2 -13494.297} C_VEL
LIN {X 0,Y 353.925,Z 448.676,A -85,B 0,C 180,E1 -13495.439,E2 -13495.439} C_VEL
LIN {X 0,Y 353.692,Z 449.735,A -85,B 0,C 180,E1 -13496.577,E2 -13496.577} C_VEL
LIN {X 0,Y 353.483,Z 450.284,A -85,B 0,C 180,E1 -13497.715,E2 -13497.715} C_VEL
LIN {X 0,Y 353.354,Z 450.323,A -85,B 0,C 180,E1 -13498.855,E2 -13498.855} C_VEL
LIN {X 0,Y 353.317,Z 449.84,A -85,B 0,C 180,E1 -13499.994,E2 -13499.994} C_VEL
LIN {X 0,Y 353.272,Z 448.747,A -85,B 0,C 180,E1 -13501.134,E2 -13501.134} C_VEL
LIN {X 0,Y 353.323,Z 446.074,A -85,B 0,C 180,E1 -13502.844,E2 -13502.844} C_VEL
LIN {X 0,Y 353.462,Z 443.551,A -85,B 0,C 180,E1 -13503.985,E2 -13503.985} C_VEL
LIN {X 0,Y 353.569,Z 438.438,A -85,B 0,C 180,E1 -13505.698,E2 -13505.698} C_VEL
LIN {X 0,Y 353.863,Z 432.908,A -85,B 0,C 180,E1 -13507.124,E2 -13507.124} C_VEL
LIN {X 0,Y 354.121,Z 427.478,A -85,B 0,C 180,E1 -13508.267,E2 -13508.267} C_VEL
LIN {X 0,Y 354.423,Z 420.935,A -85,B 0,C 180,E1 -13509.409,E2 -13509.409} C_VEL
LIN {X 0,Y 354.881,Z 411.952,A -85,B 0,C 180,E1 -13510.693,E2 -13510.693} C_VEL
LIN {X 0,Y 355.369,Z 401.596,A -85,B 0,C 180,E1 -13511.834,E2 -13511.834} C_VEL
LIN {X 0,Y 355.703,Z 393.525,A -85,B 0,C 180,E1 -13512.546,E2 -13512.546} C_VEL
LIN {X 0,Y 356.133,Z 383.303,A -85,B 0,C 180,E1 -13513.256,E2 -13513.256} C_VEL
LIN {X 0,Y 356.461,Z 371.335,A -85,B 0,C 180,E1 -13513.861,E2 -13513.861} C_VEL
LIN {X 0,Y 356.857,Z 353.516,A -85,B 0,C 180,E1 -13514.39,E2 -13514.39} C_VEL
LIN {X 0,Y 357.455,Z 309.219,A -85,B 0,C 180,E1 -13515.613,E2 -13515.613} C_VEL
LIN {X 0,Y 354.983,Z 290.867,A -85,B 0,C 180,E1 -13516.195,E2 -13516.195} C_VEL
LIN {X 0,Y 355.202,Z 283.642,A -85,B 0,C 180,E1 -13518.449,E2 -13518.449} C_VEL
LIN {X 0,Y 354.988,Z 281.077,A -85,B 0,C 180,E1 -13519.284,E2 -13519.284} C_VEL
LIN {X 0,Y 354.797,Z 281.1,A -85,B 0,C 180,E1 -13523.331,E2 -13523.331} C_VEL
LIN {X 0,Y 354.779,Z 281.102,A -85,B 0,C 180,E1 -13527.097,E2 -13527.097} C_VEL
LIN {X 0,Y 354.776,Z 281.103,A -85,B 0,C 180,E1 -13529.677,E2 -13529.677} C_VEL
LIN {X 0,Y 354.766,Z 281.108,A -85,B 0,C 180,E1 -13532.327,E2 -13532.327} C_VEL
LIN {X 0,Y 354.799,Z 281.1,A -85,B 0,C 180,E1 -13535.692,E2 -13535.692} C_VEL
LIN {X 0,Y 354.743,Z 281.107,A -85,B 0,C 180,E1 -13539.406,E2 -13539.406} C_VEL
LIN {X 0,Y 354.757,Z 281.109,A -85,B 0,C 180,E1 -13542.86,E2 -13542.86} C_VEL
LIN {X 0,Y 354.735,Z 281.108,A -85,B 0,C 180,E1 -13546.097,E2 -13546.097} C_VEL
LIN {X 0,Y 354.753,Z 281.109,A -85,B 0,C 180,E1 -13549.172,E2 -13549.172} C_VEL
LIN {X 0,Y 354.769,Z 281.105,A -85,B 0,C 180,E1 -13552.397,E2 -13552.397} C_VEL
LIN {X 0,Y 354.773,Z 281.107,A -85,B 0,C 180,E1 -13554.935,E2 -13554.935} C_VEL
LIN {X 0,Y 354.752,Z 281.106,A -85,B 0,C 180,E1 -13558.4,E2 -13558.4} C_VEL
LIN {X 0,Y 354.804,Z 281.101,A -85,B 0,C 180,E1 -13561.613,E2 -13561.613} C_VEL
LIN {X 0,Y 354.854,Z 281.093,A -85,B 0,C 180,E1 -13564.167,E2 -13564.167} C_VEL
LIN {X 0,Y 354.783,Z 281.103,A -85,B 0,C 180,E1 -13567.889,E2 -13567.889} C_VEL
LIN {X 0,Y 354.874,Z 281.093,A -85,B 0,C 180,E1 -13571.888,E2 -13571.888} C_VEL
LIN {X 0,Y 354.892,Z 281.091,A -85,B 0,C 180,E1 -13575.978,E2 -13575.978} C_VEL
LIN {X 0,Y 354.93,Z 281.088,A -85,B 0,C 180,E1 -13579.733,E2 -13579.733} C_VEL
LIN {X 0,Y 355.077,Z 281.066,A -85,B 0,C 180,E1 -13583.178,E2 -13583.178} C_VEL
LIN {X 0,Y 355.198,Z 281.054,A -85,B 0,C 180,E1 -13587.73,E2 -13587.73} C_VEL
LIN {X 0,Y 355.344,Z 281.036,A -85,B 0,C 180,E1 -13589.998,E2 -13589.998} C_VEL
LIN {X 0,Y 355.197,Z 281.054,A -85,B 0,C 180,E1 -13592.266,E2 -13592.266} C_VEL
LIN {X 0,Y 355.071,Z 281.066,A -85,B 0,C 180,E1 -13596.818,E2 -13596.818} C_VEL
LIN {X 0,Y 354.926,Z 281.088,A -85,B 0,C 180,E1 -13600.264,E2 -13600.264} C_VEL
LIN {X 0,Y 354.886,Z 281.091,A -85,B 0,C 180,E1 -13604.019,E2 -13604.019} C_VEL
LIN {X 0,Y 354.867,Z 281.094,A -85,B 0,C 180,E1 -13608.109,E2 -13608.109} C_VEL
LIN {X 0,Y 354.774,Z 281.104,A -85,B 0,C 180,E1 -13612.108,E2 -13612.108} C_VEL
LIN {X 0,Y 354.844,Z 281.094,A -85,B 0,C 180,E1 -13615.829,E2 -13615.829} C_VEL
LIN {X 0,Y 354.801,Z 281.099,A -85,B 0,C 180,E1 -13619.681,E2 -13619.681} C_VEL
LIN {X 0,Y 354.755,Z 281.105,A -85,B 0,C 180,E1 -13623.705,E2 -13623.705} C_VEL
LIN {X 0,Y 354.735,Z 281.107,A -85,B 0,C 180,E1 -13626.877,E2 -13626.877} C_VEL
LIN {X 0,Y 354.775,Z 281.106,A -85,B 0,C 180,E1 -13629.427,E2 -13629.427} C_VEL
LIN {X 0,Y 354.773,Z 281.103,A -85,B 0,C 180,E1 -13631.803,E2 -13631.803} C_VEL
LIN {X 0,Y 354.132,Z 281.186,A -85,B 0,C 180,E1 -13632.751,E2 -13632.751} C_VEL
LIN {X 0,Y 351.333,Z 281.535,A -85,B 0,C 180,E1 -13634.295,E2 -13634.295} C_VEL
LIN {X 0,Y 348.929,Z 281.836,A -85,B 0,C 180,E1 -13635.543,E2 -13635.543} C_VEL
LIN {X 0,Y 347.863,Z 281.965,A -85,B 0,C 180,E1 -13636.509,E2 -13636.509} C_VEL
LIN {X 0,Y 347.757,Z 281.976,A -85,B 0,C 180,E1 -13636.836,E2 -13636.836} C_VEL
LIN {X 0,Y 347.743,Z 281.978,A -85,B 0,C 180,E1 -13640.17,E2 -13640.17} C_VEL
LIN {X 0,Y 347.748,Z 281.978,A -85,B 0,C 180,E1 -13644.129,E2 -13644.129} C_VEL
LIN {X 0,Y 347.7,Z 281.985,A -85,B 0,C 180,E1 -13648.091,E2 -13648.091} C_VEL
LIN {X 0,Y 347.742,Z 281.979,A -85,B 0,C 180,E1 -13650.993,E2 -13650.993} C_VEL
LIN {X 0,Y 347.796,Z 281.976,A -85,B 0,C 180,E1 -13653.613,E2 -13653.613} C_VEL
LIN {X 0,Y 347.752,Z 281.98,A -85,B 0,C 180,E1 -13656.167,E2 -13656.167} C_VEL
LIN {X 0,Y 347.767,Z 281.98,A -85,B 0,C 180,E1 -13659.914,E2 -13659.914} C_VEL
LIN {X 0,Y 347.804,Z 281.972,A -85,B 0,C 180,E1 -13663.574,E2 -13663.574} C_VEL
LIN {X 0,Y 347.864,Z 281.963,A -85,B 0,C 180,E1 -13667.166,E2 -13667.166} C_VEL
LIN {X 0,Y 347.912,Z 281.959,A -85,B 0,C 180,E1 -13670.706,E2 -13670.706} C_VEL
LIN {X 0,Y 348.054,Z 281.94,A -85,B 0,C 180,E1 -13673.048,E2 -13673.048} C_VEL
LIN {X 0,Y 348.173,Z 281.925,A -85,B 0,C 180,E1 -13677.692,E2 -13677.692} C_VEL
LIN {X 0,Y 348.102,Z 281.934,A -85,B 0,C 180,E1 -13681.163,E2 -13681.163} C_VEL
LIN {X 0,Y 348.18,Z 281.928,A -85,B 0,C 180,E1 -13682.319,E2 -13682.319} C_VEL
LIN {X 0,Y 348.042,Z 281.945,A -85,B 0,C 180,E1 -13686.964,E2 -13686.964} C_VEL
LIN {X 0,Y 347.885,Z 281.964,A -85,B 0,C 180,E1 -13690.481,E2 -13690.481} C_VEL
LIN {X 0,Y 347.871,Z 281.963,A -85,B 0,C 180,E1 -13694.143,E2 -13694.143} C_VEL
LIN {X 0,Y 347.788,Z 281.973,A -85,B 0,C 180,E1 -13698.247,E2 -13698.247} C_VEL
LIN {X 0,Y 347.758,Z 281.978,A -85,B 0,C 180,E1 -13701.629,E2 -13701.629} C_VEL
LIN {X 0,Y 347.735,Z 281.984,A -85,B 0,C 180,E1 -13705.119,E2 -13705.119} C_VEL
LIN {X 0,Y 347.734,Z 281.981,A -85,B 0,C 180,E1 -13707.705,E2 -13707.705} C_VEL
LIN {X 0,Y 347.737,Z 281.979,A -85,B 0,C 180,E1 -13710.354,E2 -13710.354} C_VEL
LIN {X 0,Y 347.748,Z 281.979,A -85,B 0,C 180,E1 -13714.048,E2 -13714.048} C_VEL
LIN {X 0,Y 347.754,Z 281.981,A -85,B 0,C 180,E1 -13717.327,E2 -13717.327} C_VEL
LIN {X 0,Y 347.697,Z 281.985,A -85,B 0,C 180,E1 -13720.307,E2 -13720.307} C_VEL
LIN {X 0,Y 347.723,Z 281.984,A -85,B 0,C 180,E1 -13723.413,E2 -13723.413} C_VEL
LIN {X 0,Y 347.725,Z 281.98,A -85,B 0,C 180,E1 -13726.691,E2 -13726.691} C_VEL
LIN {X 0,Y 347.705,Z 281.986,A -85,B 0,C 180,E1 -13730.187,E2 -13730.187} C_VEL
LIN {X 0,Y 347.759,Z 281.977,A -85,B 0,C 180,E1 -13732.682,E2 -13732.682} C_VEL
LIN {X 0,Y 347.755,Z 281.981,A -85,B 0,C 180,E1 -13735.96,E2 -13735.96} C_VEL
LIN {X 0,Y 347.74,Z 281.98,A -85,B 0,C 180,E1 -13739.654,E2 -13739.654} C_VEL
LIN {X 0,Y 347.874,Z 282.05,A -85,B 0,C 180,E1 -13743.936,E2 -13743.936} C_VEL
LIN {X 0,Y 349.44,Z 291.237,A -85,B 0,C 180,E1 -13746.598,E2 -13746.598} C_VEL
LIN {X 0,Y 349.16,Z 297.176,A -85,B 0,C 180,E1 -13748.24,E2 -13748.24} C_VEL
LIN {X 0,Y 348.092,Z 310.773,A -85,B 0,C 180,E1 -13751.971,E2 -13751.971} C_VEL
LIN {X 0,Y 347.716,Z 316.759,A -85,B 0,C 180,E1 -13753.605,E2 -13753.605} C_VEL
LIN {X 0,Y 349.556,Z 337.841,A -85,B 0,C 180,E1 -13754.264,E2 -13754.264} C_VEL
LIN {X 0,Y 350.29,Z 345.892,A -85,B 0,C 180,E1 -13754.517,E2 -13754.517} C_VEL
LIN {X 0,Y 349.333,Z 395.648,A -85,B 0,C 180,E1 -13755.958,E2 -13755.958} C_VEL
LIN {X 0,Y 348.938,Z 407.823,A -85,B 0,C 180,E1 -13756.535,E2 -13756.535} C_VEL
LIN {X 0,Y 348.449,Z 417.368,A -85,B 0,C 180,E1 -13757.184,E2 -13757.184} C_VEL
LIN {X 0,Y 348.023,Z 425.779,A -85,B 0,C 180,E1 -13757.908,E2 -13757.908} C_VEL
LIN {X 0,Y 347.559,Z 433.974,A -85,B 0,C 180,E1 -13758.779,E2 -13758.779} C_VEL
LIN {X 0,Y 347.26,Z 440.813,A -85,B 0,C 180,E1 -13759.655,E2 -13759.655} C_VEL
LIN {X 0,Y 346.959,Z 447.516,A -85,B 0,C 180,E1 -13760.676,E2 -13760.676} C_VEL
LIN {X 0,Y 346.691,Z 453.896,A -85,B 0,C 180,E1 -13761.844,E2 -13761.844} C_VEL
LIN {X 0,Y 346.537,Z 459.182,A -85,B 0,C 180,E1 -13763.013,E2 -13763.013} C_VEL
LIN {X 0,Y 346.333,Z 465.51,A -85,B 0,C 180,E1 -13764.763,E2 -13764.763} C_VEL
LIN {X 0,Y 346.198,Z 470.008,A -85,B 0,C 180,E1 -13766.51,E2 -13766.51} C_VEL
LIN {X 0,Y 346.219,Z 472.272,A -85,B 0,C 180,E1 -13767.675,E2 -13767.675} C_VEL
LIN {X 0,Y 346.309,Z 473.917,A -85,B 0,C 180,E1 -13768.839,E2 -13768.839} C_VEL
LIN {X 0,Y 346.338,Z 474.911,A -85,B 0,C 180,E1 -13770.002,E2 -13770.002} C_VEL
LIN {X 0,Y 346.159,Z 475.348,A -85,B 0,C 180,E1 -13771.165,E2 -13771.165} C_VEL
LIN {X 0,Y 346.103,Z 475.277,A -85,B 0,C 180,E1 -13772.329,E2 -13772.329} C_VEL
LIN {X 0,Y 346.172,Z 474.695,A -85,B 0,C 180,E1 -13773.494,E2 -13773.494} C_VEL
LIN {X 0,Y 346.256,Z 473.553,A -85,B 0,C 180,E1 -13774.659,E2 -13774.659} C_VEL
LIN {X 0,Y 346.341,Z 471.357,A -85,B 0,C 180,E1 -13776.088,E2 -13776.088} C_VEL
LIN {X 0,Y 346.69,Z 468.132,A -85,B 0,C 180,E1 -13777.574,E2 -13777.574} C_VEL
LIN {X 0,Y 347.311,Z 462.938,A -85,B 0,C 180,E1 -13779.318,E2 -13779.318} C_VEL
LIN {X 0,Y 348.095,Z 457.408,A -85,B 0,C 180,E1 -13780.765,E2 -13780.765} C_VEL
LIN {X 0,Y 348.859,Z 452.021,A -85,B 0,C 180,E1 -13781.919,E2 -13781.919} C_VEL
LIN {X 0,Y 349.69,Z 445.585,A -85,B 0,C 180,E1 -13783.069,E2 -13783.069} C_VEL
LIN {X 0,Y 350.673,Z 437.834,A -85,B 0,C 180,E1 -13784.214,E2 -13784.214} C_VEL
LIN {X 0,Y 352.109,Z 426.889,A -85,B 0,C 180,E1 -13785.485,E2 -13785.485} C_VEL
LIN {X 0,Y 353.208,Z 417.624,A -85,B 0,C 180,E1 -13786.325,E2 -13786.325} C_VEL
LIN {X 0,Y 354.278,Z 407.865,A -85,B 0,C 180,E1 -13787.016,E2 -13787.016} C_VEL
LIN {X 0,Y 355.343,Z 396.187,A -85,B 0,C 180,E1 -13787.631,E2 -13787.631} C_VEL
LIN {X 0,Y 356.377,Z 374.352,A -85,B 0,C 180,E1 -13788.357,E2 -13788.357} C_VEL
LIN {X 0,Y 357.655,Z 347.029,A -85,B 0,C 180,E1 -13789.224,E2 -13789.224} C_VEL
LIN {X 0,Y 356.249,Z 335.182,A -85,B 0,C 180,E1 -13789.82,E2 -13789.82} C_VEL
LIN {X 0,Y 353.427,Z 321.011,A -85,B 0,C 180,E1 -13790.681,E2 -13790.681} C_VEL
LIN {X 0,Y 351.09,Z 311.465,A -85,B 0,C 180,E1 -13791.352,E2 -13791.352} C_VEL
LIN {X 0,Y 352.148,Z 299.819,A -85,B 0,C 180,E1 -13794.152,E2 -13794.152} C_VEL
LIN {X 0,Y 350.78,Z 292.789,A -85,B 0,C 180,E1 -13796.155,E2 -13796.155} C_VEL
LIN {X 0,Y 348.615,Z 284.82,A -85,B 0,C 180,E1 -13798.608,E2 -13798.608} C_VEL
LIN {X 0,Y 347.77,Z 281.982,A -85,B 0,C 180,E1 -13799.541,E2 -13799.541} C_VEL
LIN {X 0,Y 347.708,Z 281.986,A -85,B 0,C 180,E1 -13803.077,E2 -13803.077} C_VEL
LIN {X 0,Y 347.756,Z 281.979,A -85,B 0,C 180,E1 -13806.056,E2 -13806.056} C_VEL
LIN {X 0,Y 347.746,Z 281.981,A -85,B 0,C 180,E1 -13808.795,E2 -13808.795} C_VEL
LIN {X 0,Y 347.724,Z 281.98,A -85,B 0,C 180,E1 -13811.836,E2 -13811.836} C_VEL
LIN {X 0,Y 347.705,Z 281.987,A -85,B 0,C 180,E1 -13815.029,E2 -13815.029} C_VEL
LIN {X 0,Y 347.724,Z 281.98,A -85,B 0,C 180,E1 -13818.404,E2 -13818.404} C_VEL
LIN {X 0,Y 347.781,Z 281.97,A -85,B 0,C 180,E1 -13822.012,E2 -13822.012} C_VEL
LIN {X 0,Y 347.762,Z 281.976,A -85,B 0,C 180,E1 -13825.533,E2 -13825.533} C_VEL
LIN {X 0,Y 347.763,Z 281.98,A -85,B 0,C 180,E1 -13828.297,E2 -13828.297} C_VEL
LIN {X 0,Y 347.763,Z 281.979,A -85,B 0,C 180,E1 -13830.981,E2 -13830.981} C_VEL
LIN {X 0,Y 347.766,Z 281.982,A -85,B 0,C 180,E1 -13833.598,E2 -13833.598} C_VEL
LIN {X 0,Y 347.794,Z 282.032,A -85,B 0,C 180,E1 -13836.064,E2 -13836.064} C_VEL
LIN {X 0,Y 350.862,Z 291.246,A -85,B 0,C 180,E1 -13838.59,E2 -13838.59} C_VEL
LIN {X 0,Y 356.767,Z 302.978,A -85,B 0,C 180,E1 -13839.775,E2 -13839.775} C_VEL
LIN {X 0,Y 358.11,Z 306.409,A -85,B 0,C 180,E1 -13840.058,E2 -13840.058} C_VEL
LIN {X 0,Y 359.083,Z 313.95,A -85,B 0,C 180,E1 -13840.458,E2 -13840.458} C_VEL
LIN {X 0,Y 355.954,Z 373.587,A -85,B 0,C 180,E1 -13842.397,E2 -13842.397} C_VEL
LIN {X 0,Y 355.113,Z 385.414,A -85,B 0,C 180,E1 -13843.022,E2 -13843.022} C_VEL
LIN {X 0,Y 354.238,Z 395.063,A -85,B 0,C 180,E1 -13843.721,E2 -13843.721} C_VEL
LIN {X 0,Y 353.223,Z 405.577,A -85,B 0,C 180,E1 -13844.709,E2 -13844.709} C_VEL
LIN {X 0,Y 352.015,Z 414.908,A -85,B 0,C 180,E1 -13845.838,E2 -13845.838} C_VEL
LIN {X 0,Y 351.075,Z 422.467,A -85,B 0,C 180,E1 -13846.98,E2 -13846.98} C_VEL
LIN {X 0,Y 350.142,Z 428.749,A -85,B 0,C 180,E1 -13848.122,E2 -13848.122} C_VEL
LIN {X 0,Y 349.312,Z 433.98,A -85,B 0,C 180,E1 -13849.269,E2 -13849.269} C_VEL
LIN {X 0,Y 348.506,Z 439.291,A -85,B 0,C 180,E1 -13850.711,E2 -13850.711} C_VEL
LIN {X 0,Y 348.007,Z 442.691,A -85,B 0,C 180,E1 -13851.868,E2 -13851.868} C_VEL
LIN {X 0,Y 347.13,Z 446.625,A -85,B 0,C 180,E1 -13853.601,E2 -13853.601} C_VEL
LIN {X 0,Y 346.855,Z 449.224,A -85,B 0,C 180,E1 -13855.346,E2 -13855.346} C_VEL
LIN {X 0,Y 346.619,Z 450.196,A -85,B 0,C 180,E1 -13856.507,E2 -13856.507} C_VEL
LIN {X 0,Y 346.397,Z 450.633,A -85,B 0,C 180,E1 -13857.669,E2 -13857.669} C_VEL
LIN {X 0,Y 346.26,Z 450.558,A -85,B 0,C 180,E1 -13858.831,E2 -13858.831} C_VEL
LIN {X 0,Y 346.218,Z 449.966,A -85,B 0,C 180,E1 -13859.994,E2 -13859.994} C_VEL
LIN {X 0,Y 346.173,Z 448.828,A -85,B 0,C 180,E1 -13861.157,E2 -13861.157} C_VEL
LIN {X 0,Y 346.239,Z 445.957,A -85,B 0,C 180,E1 -13862.903,E2 -13862.903} C_VEL
LIN {X 0,Y 346.391,Z 443.363,A -85,B 0,C 180,E1 -13864.066,E2 -13864.066} C_VEL
LIN {X 0,Y 346.464,Z 439.094,A -85,B 0,C 180,E1 -13865.523,E2 -13865.523} C_VEL
LIN {X 0,Y 346.751,Z 433.647,A -85,B 0,C 180,E1 -13866.979,E2 -13866.979} C_VEL
LIN {X 0,Y 347.068,Z 426.803,A -85,B 0,C 180,E1 -13868.436,E2 -13868.436} C_VEL
LIN {X 0,Y 347.509,Z 418.235,A -85,B 0,C 180,E1 -13869.892,E2 -13869.892} C_VEL
LIN {X 0,Y 347.914,Z 409.455,A -85,B 0,C 180,E1 -13871.057,E2 -13871.057} C_VEL
LIN {X 0,Y 348.301,Z 401.427,A -85,B 0,C 180,E1 -13871.93,E2 -13871.93} C_VEL
LIN {X 0,Y 348.651,Z 393.261,A -85,B 0,C 180,E1 -13872.656,E2 -13872.656} C_VEL
LIN {X 0,Y 349.048,Z 384.064,A -85,B 0,C 180,E1 -13873.307,E2 -13873.307} C_VEL
LIN {X 0,Y 349.358,Z 372.378,A -85,B 0,C 180,E1 -13873.925,E2 -13873.925} C_VEL
LIN {X 0,Y 349.722,Z 356.321,A -85,B 0,C 180,E1 -13874.43,E2 -13874.43} C_VEL
LIN {X 0,Y 350.489,Z 310.268,A -85,B 0,C 180,E1 -13875.737,E2 -13875.737} C_VEL
LIN {X 0,Y 347.952,Z 291.107,A -85,B 0,C 180,E1 -13876.373,E2 -13876.373} C_VEL
LIN {X 0,Y 348.177,Z 284.615,A -85,B 0,C 180,E1 -13878.428,E2 -13878.428} C_VEL
LIN {X 0,Y 347.934,Z 281.956,A -85,B 0,C 180,E1 -13879.308,E2 -13879.308} C_VEL
LIN {X 0,Y 347.74,Z 281.982,A -85,B 0,C 180,E1 -13883.834,E2 -13883.834} C_VEL
LIN {X 0,Y 347.709,Z 281.984,A -85,B 0,C 180,E1 -13887.694,E2 -13887.694} C_VEL
LIN {X 0,Y 347.718,Z 281.986,A -85,B 0,C 180,E1 -13890.342,E2 -13890.342} C_VEL
LIN {X 0,Y 347.728,Z 281.982,A -85,B 0,C 180,E1 -13894.037,E2 -13894.037} C_VEL
LIN {X 0,Y 347.733,Z 281.98,A -85,B 0,C 180,E1 -13897.315,E2 -13897.315} C_VEL
LIN {X 0,Y 347.714,Z 281.982,A -85,B 0,C 180,E1 -13901.594,E2 -13901.594} C_VEL
LIN {X 0,Y 347.674,Z 281.99,A -85,B 0,C 180,E1 -13905.02,E2 -13905.02} C_VEL
LIN {X 0,Y 347.717,Z 281.983,A -85,B 0,C 180,E1 -13908.391,E2 -13908.391} C_VEL
LIN {X 0,Y 347.736,Z 281.979,A -85,B 0,C 180,E1 -13912.006,E2 -13912.006} C_VEL
LIN {X 0,Y 347.706,Z 281.985,A -85,B 0,C 180,E1 -13915.53,E2 -13915.53} C_VEL
LIN {X 0,Y 347.704,Z 281.983,A -85,B 0,C 180,E1 -13918.294,E2 -13918.294} C_VEL
LIN {X 0,Y 347.736,Z 281.983,A -85,B 0,C 180,E1 -13920.982,E2 -13920.982} C_VEL
LIN {X 0,Y 347.787,Z 281.976,A -85,B 0,C 180,E1 -13923.602,E2 -13923.602} C_VEL
LIN {X 0,Y 347.742,Z 281.978,A -85,B 0,C 180,E1 -13926.157,E2 -13926.157} C_VEL
LIN {X 0,Y 347.75,Z 281.979,A -85,B 0,C 180,E1 -13929.904,E2 -13929.904} C_VEL
LIN {X 0,Y 347.817,Z 281.969,A -85,B 0,C 180,E1 -13932.355,E2 -13932.355} C_VEL
LIN {X 0,Y 347.848,Z 281.968,A -85,B 0,C 180,E1 -13935.967,E2 -13935.967} C_VEL
LIN {X 0,Y 347.88,Z 281.966,A -85,B 0,C 180,E1 -13939.522,E2 -13939.522} C_VEL
LIN {X 0,Y 348.043,Z 281.941,A -85,B 0,C 180,E1 -13943.039,E2 -13943.039} C_VEL
LIN {X 0,Y 348.161,Z 281.93,A -85,B 0,C 180,E1 -13947.684,E2 -13947.684} C_VEL
LIN {X 0,Y 348.314,Z 281.912,A -85,B 0,C 180,E1 -13949.998,E2 -13949.998} C_VEL
LIN {X 0,Y 348.16,Z 281.93,A -85,B 0,C 180,E1 -13952.312,E2 -13952.312} C_VEL
LIN {X 0,Y 348.038,Z 281.942,A -85,B 0,C 180,E1 -13956.957,E2 -13956.957} C_VEL
LIN {X 0,Y 347.877,Z 281.966,A -85,B 0,C 180,E1 -13960.474,E2 -13960.474} C_VEL
LIN {X 0,Y 347.843,Z 281.97,A -85,B 0,C 180,E1 -13964.15,E2 -13964.15} C_VEL
LIN {X 0,Y 347.834,Z 281.971,A -85,B 0,C 180,E1 -13968.29,E2 -13968.29} C_VEL
LIN {X 0,Y 347.716,Z 281.986,A -85,B 0,C 180,E1 -13972.581,E2 -13972.581} C_VEL
LIN {X 0,Y 347.757,Z 281.979,A -85,B 0,C 180,E1 -13975.11,E2 -13975.11} C_VEL
LIN {X 0,Y 347.758,Z 281.976,A -85,B 0,C 180,E1 -13977.696,E2 -13977.696} C_VEL
LIN {X 0,Y 347.711,Z 281.984,A -85,B 0,C 180,E1 -13980.349,E2 -13980.349} C_VEL
LIN {X 0,Y 347.693,Z 281.986,A -85,B 0,C 180,E1 -13984.467,E2 -13984.467} C_VEL
LIN {X 0,Y 347.726,Z 281.98,A -85,B 0,C 180,E1 -13987.992,E2 -13987.992} C_VEL
LIN {X 0,Y 347.736,Z 281.98,A -85,B 0,C 180,E1 -13991.804,E2 -13991.804} C_VEL
LIN {X 0,Y 347.785,Z 281.977,A -85,B 0,C 180,E1 -13995.01,E2 -13995.01} C_VEL
LIN {X 0,Y 347.757,Z 281.976,A -85,B 0,C 180,E1 -13996.836,E2 -13996.836} C_VEL
LIN {X 0,Y 347.052,Z 282.067,A -85,B 0,C 180,E1 -13997.803,E2 -13997.803} C_VEL
LIN {X 0,Y 344.222,Z 282.422,A -85,B 0,C 180,E1 -13999.377,E2 -13999.377} C_VEL
LIN {X 0,Y 341.833,Z 282.721,A -85,B 0,C 180,E1 -14000.65,E2 -14000.65} C_VEL
LIN {X 0,Y 340.779,Z 282.85,A -85,B 0,C 180,E1 -14001.635,E2 -14001.635} C_VEL
LIN {X 0,Y 340.677,Z 282.86,A -85,B 0,C 180,E1 -14001.969,E2 -14001.969} C_VEL
LIN {X 0,Y 340.683,Z 282.863,A -85,B 0,C 180,E1 -14005.6,E2 -14005.6} C_VEL
LIN {X 0,Y 340.66,Z 282.861,A -85,B 0,C 180,E1 -14008.96,E2 -14008.96} C_VEL
LIN {X 0,Y 340.741,Z 282.851,A -85,B 0,C 180,E1 -14012.481,E2 -14012.481} C_VEL
LIN {X 0,Y 340.721,Z 282.857,A -85,B 0,C 180,E1 -14015.644,E2 -14015.644} C_VEL
LIN {X 0,Y 340.698,Z 282.858,A -85,B 0,C 180,E1 -14019.479,E2 -14019.479} C_VEL
LIN {X 0,Y 340.763,Z 282.853,A -85,B 0,C 180,E1 -14021.986,E2 -14021.986} C_VEL
LIN {X 0,Y 340.827,Z 282.842,A -85,B 0,C 180,E1 -14025.722,E2 -14025.722} C_VEL
LIN {X 0,Y 340.824,Z 282.84,A -85,B 0,C 180,E1 -14029.311,E2 -14029.311} C_VEL
LIN {X 0,Y 341.023,Z 282.816,A -85,B 0,C 180,E1 -14032.903,E2 -14032.903} C_VEL
LIN {X 0,Y 341.11,Z 282.804,A -85,B 0,C 180,E1 -14037.644,E2 -14037.644} C_VEL
LIN {X 0,Y 341.073,Z 282.81,A -85,B 0,C 180,E1 -14041.187,E2 -14041.187} C_VEL
LIN {X 0,Y 341.141,Z 282.805,A -85,B 0,C 180,E1 -14042.367,E2 -14042.367} C_VEL
LIN {X 0,Y 340.989,Z 282.822,A -85,B 0,C 180,E1 -14047.109,E2 -14047.109} C_VEL
LIN {X 0,Y 340.837,Z 282.843,A -85,B 0,C 180,E1 -14050.7,E2 -14050.7} C_VEL
LIN {X 0,Y 340.81,Z 282.843,A -85,B 0,C 180,E1 -14054.332,E2 -14054.332} C_VEL
LIN {X 0,Y 340.75,Z 282.85,A -85,B 0,C 180,E1 -14058.431,E2 -14058.431} C_VEL
LIN {X 0,Y 340.713,Z 282.854,A -85,B 0,C 180,E1 -14061.847,E2 -14061.847} C_VEL
LIN {X 0,Y 340.672,Z 282.861,A -85,B 0,C 180,E1 -14065.678,E2 -14065.678} C_VEL
LIN {X 0,Y 340.68,Z 282.858,A -85,B 0,C 180,E1 -14068.33,E2 -14068.33} C_VEL
LIN {X 0,Y 340.692,Z 282.859,A -85,B 0,C 180,E1 -14071.05,E2 -14071.05} C_VEL
LIN {X 0,Y 340.715,Z 282.858,A -85,B 0,C 180,E1 -14075.284,E2 -14075.284} C_VEL
LIN {X 0,Y 340.693,Z 282.856,A -85,B 0,C 180,E1 -14078.387,E2 -14078.387} C_VEL
LIN {X 0,Y 340.692,Z 282.859,A -85,B 0,C 180,E1 -14082.048,E2 -14082.048} C_VEL
LIN {X 0,Y 340.652,Z 282.863,A -85,B 0,C 180,E1 -14086.232,E2 -14086.232} C_VEL
LIN {X 0,Y 340.671,Z 282.859,A -85,B 0,C 180,E1 -14088.692,E2 -14088.692} C_VEL
LIN {X 0,Y 340.723,Z 282.857,A -85,B 0,C 180,E1 -14091.775,E2 -14091.775} C_VEL
LIN {X 0,Y 340.728,Z 282.854,A -85,B 0,C 180,E1 -14095.6,E2 -14095.6} C_VEL
LIN {X 0,Y 340.698,Z 282.856,A -85,B 0,C 180,E1 -14098.958,E2 -14098.958} C_VEL
LIN {X 0,Y 340.736,Z 282.851,A -85,B 0,C 180,E1 -14103.017,E2 -14103.017} C_VEL
LIN {X 0,Y 340.808,Z 282.863,A -85,B 0,C 180,E1 -14103.849,E2 -14103.849} C_VEL
LIN {X 0,Y 342.424,Z 292.646,A -85,B 0,C 180,E1 -14106.731,E2 -14106.731} C_VEL
LIN {X 0,Y 341.905,Z 300.41,A -85,B 0,C 180,E1 -14108.919,E2 -14108.919} C_VEL
LIN {X 0,Y 340.681,Z 315.759,A -85,B 0,C 180,E1 -14113.216,E2 -14113.216} C_VEL
LIN {X 0,Y 340.641,Z 316.875,A -85,B 0,C 180,E1 -14113.445,E2 -14113.445} C_VEL
LIN {X 0,Y 342.928,Z 342.651,A -85,B 0,C 180,E1 -14114.277,E2 -14114.277} C_VEL
LIN {X 0,Y 343.188,Z 346.963,A -85,B 0,C 180,E1 -14114.412,E2 -14114.412} C_VEL
LIN {X 0,Y 342.27,Z 395.223,A -85,B 0,C 180,E1 -14115.851,E2 -14115.851} C_VEL
LIN {X 0,Y 341.907,Z 406.877,A -85,B 0,C 180,E1 -14116.405,E2 -14116.405} C_VEL
LIN {X 0,Y 341.423,Z 416.56,A -85,B 0,C 180,E1 -14117.067,E2 -14117.067} C_VEL
LIN {X 0,Y 340.988,Z 425.066,A -85,B 0,C 180,E1 -14117.806,E2 -14117.806} C_VEL
LIN {X 0,Y 340.505,Z 433.335,A -85,B 0,C 180,E1 -14118.694,E2 -14118.694} C_VEL
LIN {X 0,Y 340.194,Z 440.237,A -85,B 0,C 180,E1 -14119.588,E2 -14119.588} C_VEL
LIN {X 0,Y 339.84,Z 447.855,A -85,B 0,C 180,E1 -14120.779,E2 -14120.779} C_VEL
LIN {X 0,Y 339.539,Z 455.584,A -85,B 0,C 180,E1 -14122.27,E2 -14122.27} C_VEL
LIN {X 0,Y 339.351,Z 461.701,A -85,B 0,C 180,E1 -14123.79,E2 -14123.79} C_VEL
LIN {X 0,Y 339.286,Z 466.309,A -85,B 0,C 180,E1 -14125.249,E2 -14125.249} C_VEL
LIN {X 0,Y 339.104,Z 470.498,A -85,B 0,C 180,E1 -14127.032,E2 -14127.032} C_VEL
LIN {X 0,Y 339.13,Z 471.662,A -85,B 0,C 180,E1 -14127.627,E2 -14127.627} C_VEL
LIN {X 0,Y 339.232,Z 473.352,A -85,B 0,C 180,E1 -14128.815,E2 -14128.815} C_VEL
LIN {X 0,Y 339.276,Z 474.449,A -85,B 0,C 180,E1 -14130.002,E2 -14130.002} C_VEL
LIN {X 0,Y 339.064,Z 475,A -85,B 0,C 180,E1 -14131.19,E2 -14131.19} C_VEL
LIN {X 0,Y 339.018,Z 475.044,A -85,B 0,C 180,E1 -14132.378,E2 -14132.378} C_VEL
LIN {X 0,Y 339.099,Z 474.554,A -85,B 0,C 180,E1 -14133.567,E2 -14133.567} C_VEL
LIN {X 0,Y 339.156,Z 473.44,A -85,B 0,C 180,E1 -14134.757,E2 -14134.757} C_VEL
LIN {X 0,Y 339.338,Z 470.921,A -85,B 0,C 180,E1 -14136.483,E2 -14136.483} C_VEL
LIN {X 0,Y 339.836,Z 466.778,A -85,B 0,C 180,E1 -14138.326,E2 -14138.326} C_VEL
LIN {X 0,Y 340.617,Z 461.306,A -85,B 0,C 180,E1 -14140.103,E2 -14140.103} C_VEL
LIN {X 0,Y 341.508,Z 455.469,A -85,B 0,C 180,E1 -14141.577,E2 -14141.577} C_VEL
LIN {X 0,Y 342.603,Z 448.204,A -85,B 0,C 180,E1 -14143.043,E2 -14143.043} C_VEL
LIN {X 0,Y 343.7,Z 440.065,A -85,B 0,C 180,E1 -14144.357,E2 -14144.357} C_VEL
LIN {X 0,Y 345.044,Z 431.157,A -85,B 0,C 180,E1 -14145.508,E2 -14145.508} C_VEL
LIN {X 0,Y 346.347,Z 421.546,A -85,B 0,C 180,E1 -14146.506,E2 -14146.506} C_VEL
LIN {X 0,Y 347.631,Z 410.899,A -85,B 0,C 180,E1 -14147.351,E2 -14147.351} C_VEL
LIN {X 0,Y 348.703,Z 400.239,A -85,B 0,C 180,E1 -14147.978,E2 -14147.978} C_VEL
LIN {X 0,Y 349.601,Z 388.676,A -85,B 0,C 180,E1 -14148.46,E2 -14148.46} C_VEL
LIN {X 0,Y 351.658,Z 348.275,A -85,B 0,C 180,E1 -14149.794,E2 -14149.794} C_VEL
LIN {X 0,Y 350.196,Z 336.15,A -85,B 0,C 180,E1 -14150.431,E2 -14150.431} C_VEL
LIN {X 0,Y 347.403,Z 322.077,A -85,B 0,C 180,E1 -14151.341,E2 -14151.341} C_VEL
LIN {X 0,Y 344.653,Z 311.025,A -85,B 0,C 180,E1 -14152.164,E2 -14152.164} C_VEL
LIN {X 0,Y 345.535,Z 302.314,A -85,B 0,C 180,E1 -14154.324,E2 -14154.324} C_VEL
LIN {X 0,Y 344.414,Z 296.116,A -85,B 0,C 180,E1 -14156.116,E2 -14156.116} C_VEL
LIN {X 0,Y 342.126,Z 287.482,A -85,B 0,C 180,E1 -14158.866,E2 -14158.866} C_VEL
LIN {X 0,Y 340.704,Z 282.861,A -85,B 0,C 180,E1 -14160.517,E2 -14160.517} C_VEL
LIN {X 0,Y 340.681,Z 282.862,A -85,B 0,C 180,E1 -14164.388,E2 -14164.388} C_VEL
LIN {X 0,Y 340.73,Z 282.852,A -85,B 0,C 180,E1 -14168.23,E2 -14168.23} C_VEL
LIN {X 0,Y 340.681,Z 282.858,A -85,B 0,C 180,E1 -14172.037,E2 -14172.037} C_VEL
LIN {X 0,Y 340.644,Z 282.863,A -85,B 0,C 180,E1 -14175.45,E2 -14175.45} C_VEL
LIN {X 0,Y 340.663,Z 282.861,A -85,B 0,C 180,E1 -14178.682,E2 -14178.682} C_VEL
LIN {X 0,Y 340.737,Z 282.848,A -85,B 0,C 180,E1 -14181.768,E2 -14181.768} C_VEL
LIN {X 0,Y 340.741,Z 282.85,A -85,B 0,C 180,E1 -14185.593,E2 -14185.593} C_VEL
LIN {X 0,Y 340.712,Z 282.857,A -85,B 0,C 180,E1 -14188.952,E2 -14188.952} C_VEL
LIN {X 0,Y 340.737,Z 282.859,A -85,B 0,C 180,E1 -14193.009,E2 -14193.009} C_VEL
LIN {X 0,Y 340.778,Z 282.946,A -85,B 0,C 180,E1 -14195.049,E2 -14195.049} C_VEL
LIN {X 0,Y 343.847,Z 291.896,A -85,B 0,C 180,E1 -14197.686,E2 -14197.686} C_VEL
LIN {X 0,Y 350.018,Z 303.559,A -85,B 0,C 180,E1 -14199.004,E2 -14199.004} C_VEL
LIN {X 0,Y 352.41,Z 309.308,A -85,B 0,C 180,E1 -14199.542,E2 -14199.542} C_VEL
LIN {X 0,Y 353.157,Z 315.208,A -85,B 0,C 180,E1 -14199.862,E2 -14199.862} C_VEL
LIN {X 0,Y 349.813,Z 373.366,A -85,B 0,C 180,E1 -14201.813,E2 -14201.813} C_VEL
LIN {X 0,Y 348.835,Z 385.803,A -85,B 0,C 180,E1 -14202.481,E2 -14202.481} C_VEL
LIN {X 0,Y 348.046,Z 394.566,A -85,B 0,C 180,E1 -14203.121,E2 -14203.121} C_VEL
LIN {X 0,Y 347.028,Z 403.857,A -85,B 0,C 180,E1 -14203.977,E2 -14203.977} C_VEL
LIN {X 0,Y 345.755,Z 413.762,A -85,B 0,C 180,E1 -14205.125,E2 -14205.125} C_VEL
LIN {X 0,Y 344.59,Z 422.371,A -85,B 0,C 180,E1 -14206.43,E2 -14206.43} C_VEL
LIN {X 0,Y 343.57,Z 428.677,A -85,B 0,C 180,E1 -14207.592,E2 -14207.592} C_VEL
LIN {X 0,Y 342.428,Z 435.129,A -85,B 0,C 180,E1 -14209.051,E2 -14209.051} C_VEL
LIN {X 0,Y 341.574,Z 440.302,A -85,B 0,C 180,E1 -14210.52,E2 -14210.52} C_VEL
LIN {X 0,Y 340.709,Z 445.057,A -85,B 0,C 180,E1 -14212.299,E2 -14212.299} C_VEL
LIN {X 0,Y 339.908,Z 448.257,A -85,B 0,C 180,E1 -14214.06,E2 -14214.06} C_VEL
LIN {X 0,Y 339.786,Z 449.742,A -85,B 0,C 180,E1 -14215.249,E2 -14215.249} C_VEL
LIN {X 0,Y 339.545,Z 450.66,A -85,B 0,C 180,E1 -14216.434,E2 -14216.434} C_VEL
LIN {X 0,Y 339.312,Z 450.981,A -85,B 0,C 180,E1 -14217.62,E2 -14217.62} C_VEL
LIN {X 0,Y 339.166,Z 450.788,A -85,B 0,C 180,E1 -14218.807,E2 -14218.807} C_VEL
LIN {X 0,Y 339.119,Z 450.081,A -85,B 0,C 180,E1 -14219.994,E2 -14219.994} C_VEL
LIN {X 0,Y 339.075,Z 448.846,A -85,B 0,C 180,E1 -14221.182,E2 -14221.182} C_VEL
LIN {X 0,Y 339.158,Z 445.814,A -85,B 0,C 180,E1 -14222.963,E2 -14222.963} C_VEL
LIN {X 0,Y 339.35,Z 441.439,A -85,B 0,C 180,E1 -14224.746,E2 -14224.746} C_VEL
LIN {X 0,Y 339.504,Z 435.8,A -85,B 0,C 180,E1 -14226.457,E2 -14226.457} C_VEL
LIN {X 0,Y 339.904,Z 429.013,A -85,B 0,C 180,E1 -14228.016,E2 -14228.016} C_VEL
LIN {X 0,Y 340.174,Z 422.656,A -85,B 0,C 180,E1 -14229.207,E2 -14229.207} C_VEL
LIN {X 0,Y 340.51,Z 414.95,A -85,B 0,C 180,E1 -14230.398,E2 -14230.398} C_VEL
LIN {X 0,Y 341.124,Z 405.543,A -85,B 0,C 180,E1 -14231.581,E2 -14231.581} C_VEL
LIN {X 0,Y 341.519,Z 394.765,A -85,B 0,C 180,E1 -14232.623,E2 -14232.623} C_VEL
LIN {X 0,Y 341.957,Z 384.806,A -85,B 0,C 180,E1 -14233.362,E2 -14233.362} C_VEL
LIN {X 0,Y 342.263,Z 374.848,A -85,B 0,C 180,E1 -14233.917,E2 -14233.917} C_VEL
LIN {X 0,Y 342.562,Z 360.499,A -85,B 0,C 180,E1 -14234.435,E2 -14234.435} C_VEL
LIN {X 0,Y 343.436,Z 310.672,A -85,B 0,C 180,E1 -14235.884,E2 -14235.884} C_VEL
LIN {X 0,Y 340.926,Z 291.396,A -85,B 0,C 180,E1 -14236.536,E2 -14236.536} C_VEL
LIN {X 0,Y 341.12,Z 284.97,A -85,B 0,C 180,E1 -14238.604,E2 -14238.604} C_VEL
LIN {X 0,Y 340.887,Z 282.833,A -85,B 0,C 180,E1 -14239.332,E2 -14239.332} C_VEL
LIN {X 0,Y 340.694,Z 282.856,A -85,B 0,C 180,E1 -14243.068,E2 -14243.068} C_VEL
LIN {X 0,Y 340.696,Z 282.856,A -85,B 0,C 180,E1 -14246.981,E2 -14246.981} C_VEL
LIN {X 0,Y 340.673,Z 282.859,A -85,B 0,C 180,E1 -14251.038,E2 -14251.038} C_VEL
LIN {X 0,Y 340.696,Z 282.856,A -85,B 0,C 180,E1 -14255.272,E2 -14255.272} C_VEL
LIN {X 0,Y 340.669,Z 282.863,A -85,B 0,C 180,E1 -14258.375,E2 -14258.375} C_VEL
LIN {X 0,Y 340.666,Z 282.86,A -85,B 0,C 180,E1 -14262.037,E2 -14262.037} C_VEL
LIN {X 0,Y 340.621,Z 282.866,A -85,B 0,C 180,E1 -14266.22,E2 -14266.22} C_VEL
LIN {X 0,Y 340.653,Z 282.861,A -85,B 0,C 180,E1 -14269.747,E2 -14269.747} C_VEL
LIN {X 0,Y 340.667,Z 282.863,A -85,B 0,C 180,E1 -14273.252,E2 -14273.252} C_VEL
LIN {X 0,Y 340.654,Z 282.861,A -85,B 0,C 180,E1 -14276.147,E2 -14276.147} C_VEL
LIN {X 0,Y 340.696,Z 282.856,A -85,B 0,C 180,E1 -14280.323,E2 -14280.323} C_VEL
LIN {X 0,Y 340.748,Z 282.853,A -85,B 0,C 180,E1 -14283.013,E2 -14283.013} C_VEL
LIN {X 0,Y 340.711,Z 282.857,A -85,B 0,C 180,E1 -14285.633,E2 -14285.633} C_VEL
LIN {X 0,Y 340.684,Z 282.863,A -85,B 0,C 180,E1 -14289.468,E2 -14289.468} C_VEL
LIN {X 0,Y 340.809,Z 282.844,A -85,B 0,C 180,E1 -14291.98,E2 -14291.98} C_VEL
LIN {X 0,Y 340.82,Z 282.846,A -85,B 0,C 180,E1 -14295.701,E2 -14295.701} C_VEL
LIN {X 0,Y 340.823,Z 282.842,A -85,B 0,C 180,E1 -14299.303,E2 -14299.303} C_VEL
LIN {X 0,Y 341.01,Z 282.817,A -85,B 0,C 180,E1 -14302.895,E2 -14302.895} C_VEL
LIN {X 0,Y 341.124,Z 282.806,A -85,B 0,C 180,E1 -14307.636,E2 -14307.636} C_VEL
LIN {X 0,Y 341.263,Z 282.79,A -85,B 0,C 180,E1 -14309.998,E2 -14309.998} C_VEL
LIN {X 0,Y 341.122,Z 282.806,A -85,B 0,C 180,E1 -14312.36,E2 -14312.36} C_VEL
LIN {X 0,Y 341.006,Z 282.817,A -85,B 0,C 180,E1 -14317.101,E2 -14317.101} C_VEL
LIN {X 0,Y 340.819,Z 282.843,A -85,B 0,C 180,E1 -14320.693,E2 -14320.693} C_VEL
LIN {X 0,Y 340.808,Z 282.847,A -85,B 0,C 180,E1 -14324.325,E2 -14324.325} C_VEL
LIN {X 0,Y 340.78,Z 282.85,A -85,B 0,C 180,E1 -14328.466,E2 -14328.466} C_VEL
LIN {X 0,Y 340.667,Z 282.86,A -85,B 0,C 180,E1 -14331.845,E2 -14331.845} C_VEL
LIN {X 0,Y 340.718,Z 282.853,A -85,B 0,C 180,E1 -14335.666,E2 -14335.666} C_VEL
LIN {X 0,Y 340.689,Z 282.859,A -85,B 0,C 180,E1 -14338.322,E2 -14338.322} C_VEL
LIN {X 0,Y 340.651,Z 282.866,A -85,B 0,C 180,E1 -14341.047,E2 -14341.047} C_VEL
LIN {X 0,Y 340.667,Z 282.863,A -85,B 0,C 180,E1 -14345.282,E2 -14345.282} C_VEL
LIN {X 0,Y 340.668,Z 282.86,A -85,B 0,C 180,E1 -14348.391,E2 -14348.391} C_VEL
LIN {X 0,Y 340.678,Z 282.863,A -85,B 0,C 180,E1 -14351.307,E2 -14351.307} C_VEL
LIN {X 0,Y 340.735,Z 282.851,A -85,B 0,C 180,E1 -14354.526,E2 -14354.526} C_VEL
LIN {X 0,Y 340.707,Z 282.855,A -85,B 0,C 180,E1 -14357.949,E2 -14357.949} C_VEL
LIN {X 0,Y 340.691,Z 282.856,A -85,B 0,C 180,E1 -14360.257,E2 -14360.257} C_VEL
LIN {X 0,Y 340.677,Z 282.86,A -85,B 0,C 180,E1 -14361.969,E2 -14361.969} C_VEL
LIN {X 0,Y 339.96,Z 282.951,A -85,B 0,C 180,E1 -14362.956,E2 -14362.956} C_VEL
LIN {X 0,Y 337.081,Z 283.306,A -85,B 0,C 180,E1 -14364.562,E2 -14364.562} C_VEL
LIN {X 0,Y 334.682,Z 283.608,A -85,B 0,C 180,E1 -14365.863,E2 -14365.863} C_VEL
LIN {X 0,Y 333.672,Z 283.732,A -85,B 0,C 180,E1 -14366.87,E2 -14366.87} C_VEL
LIN {X 0,Y 333.598,Z 283.742,A -85,B 0,C 180,E1 -14367.211,E2 -14367.211} C_VEL
LIN {X 0,Y 333.654,Z 283.733,A -85,B 0,C 180,E1 -14371.031,E2 -14371.031} C_VEL
LIN {X 0,Y 333.7,Z 283.733,A -85,B 0,C 180,E1 -14373.759,E2 -14373.759} C_VEL
LIN {X 0,Y 333.625,Z 283.741,A -85,B 0,C 180,E1 -14377.725,E2 -14377.725} C_VEL
LIN {X 0,Y 333.712,Z 283.728,A -85,B 0,C 180,E1 -14381.592,E2 -14381.592} C_VEL
LIN {X 0,Y 333.782,Z 283.718,A -85,B 0,C 180,E1 -14385.583,E2 -14385.583} C_VEL
LIN {X 0,Y 333.793,Z 283.715,A -85,B 0,C 180,E1 -14389.084,E2 -14389.084} C_VEL
LIN {X 0,Y 333.97,Z 283.695,A -85,B 0,C 180,E1 -14392.753,E2 -14392.753} C_VEL
LIN {X 0,Y 333.77,Z 283.719,A -85,B 0,C 180,E1 -14395.175,E2 -14395.175} C_VEL
LIN {X 0,Y 334.051,Z 283.683,A -85,B 0,C 180,E1 -14397.595,E2 -14397.595} C_VEL
LIN {X 0,Y 334.044,Z 283.685,A -85,B 0,C 180,E1 -14401.212,E2 -14401.212} C_VEL
LIN {X 0,Y 334.078,Z 283.685,A -85,B 0,C 180,E1 -14402.417,E2 -14402.417} C_VEL
LIN {X 0,Y 333.977,Z 283.693,A -85,B 0,C 180,E1 -14406.045,E2 -14406.045} C_VEL
LIN {X 0,Y 333.809,Z 283.713,A -85,B 0,C 180,E1 -14409.702,E2 -14409.702} C_VEL
LIN {X 0,Y 333.777,Z 283.719,A -85,B 0,C 180,E1 -14413.398,E2 -14413.398} C_VEL
LIN {X 0,Y 333.678,Z 283.734,A -85,B 0,C 180,E1 -14417.155,E2 -14417.155} C_VEL
LIN {X 0,Y 333.645,Z 283.735,A -85,B 0,C 180,E1 -14419.701,E2 -14419.701} C_VEL
LIN {X 0,Y 333.644,Z 283.734,A -85,B 0,C 180,E1 -14422.287,E2 -14422.287} C_VEL
LIN {X 0,Y 333.655,Z 283.738,A -85,B 0,C 180,E1 -14425.084,E2 -14425.084} C_VEL
LIN {X 0,Y 333.651,Z 283.736,A -85,B 0,C 180,E1 -14428.983,E2 -14428.983} C_VEL
LIN {X 0,Y 333.643,Z 283.734,A -85,B 0,C 180,E1 -14432.592,E2 -14432.592} C_VEL
LIN {X 0,Y 333.673,Z 283.731,A -85,B 0,C 180,E1 -14436.144,E2 -14436.144} C_VEL
LIN {X 0,Y 333.602,Z 283.742,A -85,B 0,C 180,E1 -14439.204,E2 -14439.204} C_VEL
LIN {X 0,Y 333.628,Z 283.736,A -85,B 0,C 180,E1 -14442.503,E2 -14442.503} C_VEL
LIN {X 0,Y 333.596,Z 283.744,A -85,B 0,C 180,E1 -14445.959,E2 -14445.959} C_VEL
LIN {X 0,Y 333.606,Z 283.74,A -85,B 0,C 180,E1 -14449.329,E2 -14449.329} C_VEL
LIN {X 0,Y 333.666,Z 283.731,A -85,B 0,C 180,E1 -14453.173,E2 -14453.173} C_VEL
LIN {X 0,Y 333.678,Z 283.73,A -85,B 0,C 180,E1 -14455.345,E2 -14455.345} C_VEL
LIN {X 0,Y 333.635,Z 283.74,A -85,B 0,C 180,E1 -14458.225,E2 -14458.225} C_VEL
LIN {X 0,Y 333.632,Z 283.736,A -85,B 0,C 180,E1 -14461.023,E2 -14461.023} C_VEL
LIN {X 0,Y 333.801,Z 283.909,A -85,B 0,C 180,E1 -14463.832,E2 -14463.832} C_VEL
LIN {X 0,Y 335.332,Z 292.874,A -85,B 0,C 180,E1 -14466.536,E2 -14466.536} C_VEL
LIN {X 0,Y 335.045,Z 298.442,A -85,B 0,C 180,E1 -14468.143,E2 -14468.143} C_VEL
LIN {X 0,Y 333.92,Z 311.601,A -85,B 0,C 180,E1 -14471.917,E2 -14471.917} C_VEL
LIN {X 0,Y 333.599,Z 316.246,A -85,B 0,C 180,E1 -14473.243,E2 -14473.243} C_VEL
LIN {X 0,Y 334.786,Z 332.022,A -85,B 0,C 180,E1 -14473.782,E2 -14473.782} C_VEL
LIN {X 0,Y 336.156,Z 347.031,A -85,B 0,C 180,E1 -14474.273,E2 -14474.273} C_VEL
LIN {X 0,Y 335.204,Z 395.5,A -85,B 0,C 180,E1 -14475.779,E2 -14475.779} C_VEL
LIN {X 0,Y 334.783,Z 407.968,A -85,B 0,C 180,E1 -14476.419,E2 -14476.419} C_VEL
LIN {X 0,Y 334.293,Z 417.31,A -85,B 0,C 180,E1 -14477.095,E2 -14477.095} C_VEL
LIN {X 0,Y 333.836,Z 425.588,A -85,B 0,C 180,E1 -14477.849,E2 -14477.849} C_VEL
LIN {X 0,Y 333.391,Z 433.704,A -85,B 0,C 180,E1 -14478.758,E2 -14478.758} C_VEL
LIN {X 0,Y 333.069,Z 441.532,A -85,B 0,C 180,E1 -14479.824,E2 -14479.824} C_VEL
LIN {X 0,Y 332.685,Z 449.761,A -85,B 0,C 180,E1 -14481.192,E2 -14481.192} C_VEL
LIN {X 0,Y 332.417,Z 456.911,A -85,B 0,C 180,E1 -14482.714,E2 -14482.714} C_VEL
LIN {X 0,Y 332.221,Z 462.881,A -85,B 0,C 180,E1 -14484.329,E2 -14484.329} C_VEL
LIN {X 0,Y 332.15,Z 467.025,A -85,B 0,C 180,E1 -14485.755,E2 -14485.755} C_VEL
LIN {X 0,Y 332.029,Z 469.781,A -85,B 0,C 180,E1 -14486.969,E2 -14486.969} C_VEL
LIN {X 0,Y 332.157,Z 472.767,A -85,B 0,C 180,E1 -14488.79,E2 -14488.79} C_VEL
LIN {X 0,Y 332.214,Z 473.986,A -85,B 0,C 180,E1 -14490.002,E2 -14490.002} C_VEL
LIN {X 0,Y 331.97,Z 474.652,A -85,B 0,C 180,E1 -14491.215,E2 -14491.215} C_VEL
LIN {X 0,Y 331.935,Z 474.809,A -85,B 0,C 180,E1 -14492.429,E2 -14492.429} C_VEL
LIN {X 0,Y 332.027,Z 474.366,A -85,B 0,C 180,E1 -14493.643,E2 -14493.643} C_VEL
LIN {X 0,Y 332.062,Z 473.337,A -85,B 0,C 180,E1 -14494.858,E2 -14494.858} C_VEL
LIN {X 0,Y 332.285,Z 470.878,A -85,B 0,C 180,E1 -14496.682,E2 -14496.682} C_VEL
LIN {X 0,Y 332.817,Z 467.054,A -85,B 0,C 180,E1 -14498.502,E2 -14498.502} C_VEL
LIN {X 0,Y 333.486,Z 462.734,A -85,B 0,C 180,E1 -14500.014,E2 -14500.014} C_VEL
LIN {X 0,Y 334.419,Z 457.317,A -85,B 0,C 180,E1 -14501.518,E2 -14501.518} C_VEL
LIN {X 0,Y 335.537,Z 450.601,A -85,B 0,C 180,E1 -14503.014,E2 -14503.014} C_VEL
LIN {X 0,Y 336.797,Z 442.308,A -85,B 0,C 180,E1 -14504.503,E2 -14504.503} C_VEL
LIN {X 0,Y 338.353,Z 432.723,A -85,B 0,C 180,E1 -14505.822,E2 -14505.822} C_VEL
LIN {X 0,Y 339.675,Z 423.499,A -85,B 0,C 180,E1 -14506.84,E2 -14506.84} C_VEL
LIN {X 0,Y 340.987,Z 413.772,A -85,B 0,C 180,E1 -14507.7,E2 -14507.7} C_VEL
LIN {X 0,Y 342.423,Z 401.247,A -85,B 0,C 180,E1 -14508.513,E2 -14508.513} C_VEL
LIN {X 0,Y 343.394,Z 390.374,A -85,B 0,C 180,E1 -14509,E2 -14509} C_VEL
LIN {X 0,Y 345.643,Z 348.612,A -85,B 0,C 180,E1 -14510.43,E2 -14510.43} C_VEL
LIN {X 0,Y 344.281,Z 337.498,A -85,B 0,C 180,E1 -14511.063,E2 -14511.063} C_VEL
LIN {X 0,Y 341.725,Z 324.295,A -85,B 0,C 180,E1 -14511.956,E2 -14511.956} C_VEL
LIN {X 0,Y 338.351,Z 310.512,A -85,B 0,C 180,E1 -14513.069,E2 -14513.069} C_VEL
LIN {X 0,Y 338.929,Z 303.626,A -85,B 0,C 180,E1 -14514.83,E2 -14514.83} C_VEL
LIN {X 0,Y 336.861,Z 294.378,A -85,B 0,C 180,E1 -14517.736,E2 -14517.736} C_VEL
LIN {X 0,Y 334.527,Z 286.477,A -85,B 0,C 180,E1 -14520.524,E2 -14520.524} C_VEL
LIN {X 0,Y 333.626,Z 283.741,A -85,B 0,C 180,E1 -14521.603,E2 -14521.603} C_VEL
LIN {X 0,Y 333.636,Z 283.738,A -85,B 0,C 180,E1 -14524.756,E2 -14524.756} C_VEL
LIN {X 0,Y 333.652,Z 283.736,A -85,B 0,C 180,E1 -14527.653,E2 -14527.653} C_VEL
LIN {X 0,Y 333.616,Z 283.742,A -85,B 0,C 180,E1 -14530.774,E2 -14530.774} C_VEL
LIN {X 0,Y 333.597,Z 283.741,A -85,B 0,C 180,E1 -14534.246,E2 -14534.246} C_VEL
LIN {X 0,Y 333.633,Z 283.734,A -85,B 0,C 180,E1 -14537.612,E2 -14537.612} C_VEL
LIN {X 0,Y 333.635,Z 283.735,A -85,B 0,C 180,E1 -14541.208,E2 -14541.208} C_VEL
LIN {X 0,Y 333.692,Z 283.726,A -85,B 0,C 180,E1 -14543.858,E2 -14543.858} C_VEL
LIN {X 0,Y 333.663,Z 283.733,A -85,B 0,C 180,E1 -14547.41,E2 -14547.41} C_VEL
LIN {X 0,Y 333.671,Z 283.735,A -85,B 0,C 180,E1 -14551.019,E2 -14551.019} C_VEL
LIN {X 0,Y 333.686,Z 283.819,A -85,B 0,C 180,E1 -14553.865,E2 -14553.865} C_VEL
LIN {X 0,Y 336.886,Z 292.609,A -85,B 0,C 180,E1 -14556.699,E2 -14556.699} C_VEL
LIN {X 0,Y 343.118,Z 303.889,A -85,B 0,C 180,E1 -14558.137,E2 -14558.137} C_VEL
LIN {X 0,Y 346.825,Z 312.112,A -85,B 0,C 180,E1 -14558.974,E2 -14558.974} C_VEL
LIN {X 0,Y 347.274,Z 316.947,A -85,B 0,C 180,E1 -14559.238,E2 -14559.238} C_VEL
LIN {X 0,Y 343.688,Z 374.649,A -85,B 0,C 180,E1 -14561.246,E2 -14561.246} C_VEL
LIN {X 0,Y 342.663,Z 386.688,A -85,B 0,C 180,E1 -14561.923,E2 -14561.923} C_VEL
LIN {X 0,Y 341.703,Z 396.084,A -85,B 0,C 180,E1 -14562.644,E2 -14562.644} C_VEL
LIN {X 0,Y 340.442,Z 406.457,A -85,B 0,C 180,E1 -14563.659,E2 -14563.659} C_VEL
LIN {X 0,Y 338.932,Z 416.675,A -85,B 0,C 180,E1 -14564.972,E2 -14564.972} C_VEL
LIN {X 0,Y 337.843,Z 424.026,A -85,B 0,C 180,E1 -14566.154,E2 -14566.154} C_VEL
LIN {X 0,Y 336.789,Z 430.129,A -85,B 0,C 180,E1 -14567.338,E2 -14567.338} C_VEL
LIN {X 0,Y 335.588,Z 436.395,A -85,B 0,C 180,E1 -14568.825,E2 -14568.825} C_VEL
LIN {X 0,Y 334.65,Z 441.356,A -85,B 0,C 180,E1 -14570.322,E2 -14570.322} C_VEL
LIN {X 0,Y 333.685,Z 445.954,A -85,B 0,C 180,E1 -14572.213,E2 -14572.213} C_VEL
LIN {X 0,Y 332.881,Z 448.876,A -85,B 0,C 180,E1 -14573.935,E2 -14573.935} C_VEL
LIN {X 0,Y 332.716,Z 450.236,A -85,B 0,C 180,E1 -14575.147,E2 -14575.147} C_VEL
LIN {X 0,Y 332.47,Z 451.088,A -85,B 0,C 180,E1 -14576.358,E2 -14576.358} C_VEL
LIN {X 0,Y 332.227,Z 451.342,A -85,B 0,C 180,E1 -14577.569,E2 -14577.569} C_VEL
LIN {X 0,Y 332.071,Z 451.016,A -85,B 0,C 180,E1 -14578.781,E2 -14578.781} C_VEL
LIN {X 0,Y 332.02,Z 450.179,A -85,B 0,C 180,E1 -14579.994,E2 -14579.994} C_VEL
LIN {X 0,Y 331.98,Z 448.824,A -85,B 0,C 180,E1 -14581.207,E2 -14581.207} C_VEL
LIN {X 0,Y 332.03,Z 446.923,A -85,B 0,C 180,E1 -14582.42,E2 -14582.42} C_VEL
LIN {X 0,Y 332.168,Z 444.379,A -85,B 0,C 180,E1 -14583.633,E2 -14583.633} C_VEL
LIN {X 0,Y 332.273,Z 439.227,A -85,B 0,C 180,E1 -14585.455,E2 -14585.455} C_VEL
LIN {X 0,Y 332.541,Z 434.221,A -85,B 0,C 180,E1 -14586.837,E2 -14586.837} C_VEL
LIN {X 0,Y 332.838,Z 428.2,A -85,B 0,C 180,E1 -14588.188,E2 -14588.188} C_VEL
LIN {X 0,Y 333.134,Z 421.621,A -85,B 0,C 180,E1 -14589.403,E2 -14589.403} C_VEL
LIN {X 0,Y 333.63,Z 412.606,A -85,B 0,C 180,E1 -14590.768,E2 -14590.768} C_VEL
LIN {X 0,Y 334.069,Z 403.71,A -85,B 0,C 180,E1 -14591.829,E2 -14591.829} C_VEL
LIN {X 0,Y 334.46,Z 394.128,A -85,B 0,C 180,E1 -14592.739,E2 -14592.739} C_VEL
LIN {X 0,Y 334.857,Z 385.082,A -85,B 0,C 180,E1 -14593.418,E2 -14593.418} C_VEL
LIN {X 0,Y 335.182,Z 374.462,A -85,B 0,C 180,E1 -14594.024,E2 -14594.024} C_VEL
LIN {X 0,Y 335.522,Z 359.963,A -85,B 0,C 180,E1 -14594.551,E2 -14594.551} C_VEL
LIN {X 0,Y 336.379,Z 311.131,A -85,B 0,C 180,E1 -14596.033,E2 -14596.033} C_VEL
LIN {X 0,Y 333.879,Z 291.649,A -85,B 0,C 180,E1 -14596.698,E2 -14596.698} C_VEL
LIN {X 0,Y 334.024,Z 285.363,A -85,B 0,C 180,E1 -14598.766,E2 -14598.766} C_VEL
LIN {X 0,Y 333.843,Z 283.711,A -85,B 0,C 180,E1 -14599.349,E2 -14599.349} C_VEL
LIN {X 0,Y 333.633,Z 283.737,A -85,B 0,C 180,E1 -14603.585,E2 -14603.585} C_VEL
LIN {X 0,Y 333.643,Z 283.735,A -85,B 0,C 180,E1 -14607.599,E2 -14607.599} C_VEL
LIN {X 0,Y 333.639,Z 283.74,A -85,B 0,C 180,E1 -14610.359,E2 -14610.359} C_VEL
LIN {X 0,Y 333.617,Z 283.738,A -85,B 0,C 180,E1 -14613.201,E2 -14613.201} C_VEL
LIN {X 0,Y 333.653,Z 283.735,A -85,B 0,C 180,E1 -14616.132,E2 -14616.132} C_VEL
LIN {X 0,Y 333.577,Z 283.743,A -85,B 0,C 180,E1 -14619.192,E2 -14619.192} C_VEL
LIN {X 0,Y 333.601,Z 283.744,A -85,B 0,C 180,E1 -14622.492,E2 -14622.492} C_VEL
LIN {X 0,Y 333.565,Z 283.744,A -85,B 0,C 180,E1 -14625.948,E2 -14625.948} C_VEL
LIN {X 0,Y 333.614,Z 283.74,A -85,B 0,C 180,E1 -14629.309,E2 -14629.309} C_VEL
LIN {X 0,Y 333.628,Z 283.74,A -85,B 0,C 180,E1 -14633.162,E2 -14633.162} C_VEL
LIN {X 0,Y 333.636,Z 283.738,A -85,B 0,C 180,E1 -14635.335,E2 -14635.335} C_VEL
LIN {X 0,Y 333.59,Z 283.741,A -85,B 0,C 180,E1 -14638.216,E2 -14638.216} C_VEL
LIN {X 0,Y 333.67,Z 283.731,A -85,B 0,C 180,E1 -14642.187,E2 -14642.187} C_VEL
LIN {X 0,Y 333.682,Z 283.733,A -85,B 0,C 180,E1 -14645.085,E2 -14645.085} C_VEL
LIN {X 0,Y 333.625,Z 283.739,A -85,B 0,C 180,E1 -14649.014,E2 -14649.014} C_VEL
LIN {X 0,Y 333.745,Z 283.727,A -85,B 0,C 180,E1 -14651.585,E2 -14651.585} C_VEL
LIN {X 0,Y 333.759,Z 283.725,A -85,B 0,C 180,E1 -14655.573,E2 -14655.573} C_VEL
LIN {X 0,Y 333.786,Z 283.717,A -85,B 0,C 180,E1 -14659.075,E2 -14659.075} C_VEL
LIN {X 0,Y 333.962,Z 283.694,A -85,B 0,C 180,E1 -14662.744,E2 -14662.744} C_VEL
LIN {X 0,Y 333.765,Z 283.719,A -85,B 0,C 180,E1 -14665.166,E2 -14665.166} C_VEL
LIN {X 0,Y 334.086,Z 283.682,A -85,B 0,C 180,E1 -14667.587,E2 -14667.587} C_VEL
LIN {X 0,Y 334.213,Z 283.669,A -85,B 0,C 180,E1 -14669.998,E2 -14669.998} C_VEL
LIN {X 0,Y 334.084,Z 283.682,A -85,B 0,C 180,E1 -14672.409,E2 -14672.409} C_VEL
LIN {X 0,Y 333.958,Z 283.695,A -85,B 0,C 180,E1 -14677.252,E2 -14677.252} C_VEL
LIN {X 0,Y 333.782,Z 283.718,A -85,B 0,C 180,E1 -14680.921,E2 -14680.921} C_VEL
LIN {X 0,Y 333.753,Z 283.724,A -85,B 0,C 180,E1 -14684.634,E2 -14684.634} C_VEL
LIN {X 0,Y 333.739,Z 283.727,A -85,B 0,C 180,E1 -14688.654,E2 -14688.654} C_VEL
LIN {X 0,Y 333.607,Z 283.741,A -85,B 0,C 180,E1 -14692.282,E2 -14692.282} C_VEL
LIN {X 0,Y 333.682,Z 283.731,A -85,B 0,C 180,E1 -14696.248,E2 -14696.248} C_VEL
LIN {X 0,Y 333.658,Z 283.737,A -85,B 0,C 180,E1 -14698.974,E2 -14698.974} C_VEL
LIN {X 0,Y 333.592,Z 283.744,A -85,B 0,C 180,E1 -14702.589,E2 -14702.589} C_VEL
LIN {X 0,Y 333.626,Z 283.736,A -85,B 0,C 180,E1 -14706.142,E2 -14706.142} C_VEL
LIN {X 0,Y 333.635,Z 283.74,A -85,B 0,C 180,E1 -14709.191,E2 -14709.191} C_VEL
LIN {X 0,Y 333.656,Z 283.733,A -85,B 0,C 180,E1 -14712.517,E2 -14712.517} C_VEL
LIN {X 0,Y 333.684,Z 283.73,A -85,B 0,C 180,E1 -14715.981,E2 -14715.981} C_VEL
LIN {X 0,Y 333.659,Z 283.738,A -85,B 0,C 180,E1 -14719.309,E2 -14719.309} C_VEL
LIN {X 0,Y 333.625,Z 283.74,A -85,B 0,C 180,E1 -14723.173,E2 -14723.173} C_VEL
LIN {X 0,Y 333.634,Z 283.74,A -85,B 0,C 180,E1 -14725.346,E2 -14725.346} C_VEL
LIN {X 0,Y 333.598,Z 283.742,A -85,B 0,C 180,E1 -14727.211,E2 -14727.211} C_VEL
LIN {X 0,Y 332.953,Z 283.828,A -85,B 0,C 180,E1 -14728.218,E2 -14728.218} C_VEL
LIN {X 0,Y 330.114,Z 284.183,A -85,B 0,C 180,E1 -14729.859,E2 -14729.859} C_VEL
LIN {X 0,Y 327.707,Z 284.478,A -85,B 0,C 180,E1 -14731.187,E2 -14731.187} C_VEL
LIN {X 0,Y 326.69,Z 284.602,A -85,B 0,C 180,E1 -14732.216,E2 -14732.216} C_VEL
LIN {X 0,Y 326.616,Z 284.609,A -85,B 0,C 180,E1 -14732.564,E2 -14732.564} C_VEL
LIN {X 0,Y 326.616,Z 284.615,A -85,B 0,C 180,E1 -14735.877,E2 -14735.877} C_VEL
LIN {X 0,Y 326.592,Z 284.618,A -85,B 0,C 180,E1 -14739.868,E2 -14739.868} C_VEL
LIN {X 0,Y 326.691,Z 284.603,A -85,B 0,C 180,E1 -14743.767,E2 -14743.767} C_VEL
LIN {X 0,Y 326.731,Z 284.599,A -85,B 0,C 180,E1 -14746.321,E2 -14746.321} C_VEL
LIN {X 0,Y 326.76,Z 284.596,A -85,B 0,C 180,E1 -14750.099,E2 -14750.099} C_VEL
LIN {X 0,Y 326.939,Z 284.571,A -85,B 0,C 180,E1 -14753.836,E2 -14753.836} C_VEL
LIN {X 0,Y 326.994,Z 284.562,A -85,B 0,C 180,E1 -14757.543,E2 -14757.543} C_VEL
LIN {X 0,Y 327.015,Z 284.56,A -85,B 0,C 180,E1 -14761.238,E2 -14761.238} C_VEL
LIN {X 0,Y 327.018,Z 284.564,A -85,B 0,C 180,E1 -14762.47,E2 -14762.47} C_VEL
LIN {X 0,Y 326.931,Z 284.572,A -85,B 0,C 180,E1 -14766.176,E2 -14766.176} C_VEL
LIN {X 0,Y 326.772,Z 284.59,A -85,B 0,C 180,E1 -14769.913,E2 -14769.913} C_VEL
LIN {X 0,Y 326.734,Z 284.595,A -85,B 0,C 180,E1 -14773.692,E2 -14773.692} C_VEL
LIN {X 0,Y 326.624,Z 284.609,A -85,B 0,C 180,E1 -14777.537,E2 -14777.537} C_VEL
LIN {X 0,Y 326.6,Z 284.611,A -85,B 0,C 180,E1 -14780.144,E2 -14780.144} C_VEL
LIN {X 0,Y 326.586,Z 284.616,A -85,B 0,C 180,E1 -14782.795,E2 -14782.795} C_VEL
LIN {X 0,Y 326.6,Z 284.614,A -85,B 0,C 180,E1 -14786.87,E2 -14786.87} C_VEL
LIN {X 0,Y 326.61,Z 284.61,A -85,B 0,C 180,E1 -14790.608,E2 -14790.608} C_VEL
LIN {X 0,Y 326.606,Z 284.612,A -85,B 0,C 180,E1 -14794.025,E2 -14794.025} C_VEL
LIN {X 0,Y 326.622,Z 284.612,A -85,B 0,C 180,E1 -14797.242,E2 -14797.242} C_VEL
LIN {X 0,Y 326.545,Z 284.62,A -85,B 0,C 180,E1 -14801.129,E2 -14801.129} C_VEL
LIN {X 0,Y 326.56,Z 284.621,A -85,B 0,C 180,E1 -14803.531,E2 -14803.531} C_VEL
LIN {X 0,Y 326.575,Z 284.615,A -85,B 0,C 180,E1 -14807.034,E2 -14807.034} C_VEL
LIN {X 0,Y 326.576,Z 284.614,A -85,B 0,C 180,E1 -14810.786,E2 -14810.786} C_VEL
LIN {X 0,Y 326.616,Z 284.611,A -85,B 0,C 180,E1 -14814.484,E2 -14814.484} C_VEL
LIN {X 0,Y 326.613,Z 284.61,A -85,B 0,C 180,E1 -14817.459,E2 -14817.459} C_VEL
LIN {X 0,Y 326.585,Z 284.618,A -85,B 0,C 180,E1 -14820.336,E2 -14820.336} C_VEL
LIN {X 0,Y 326.736,Z 284.706,A -85,B 0,C 180,E1 -14823.753,E2 -14823.753} C_VEL
LIN {X 0,Y 328.295,Z 293.863,A -85,B 0,C 180,E1 -14826.569,E2 -14826.569} C_VEL
LIN {X 0,Y 327.708,Z 301.935,A -85,B 0,C 180,E1 -14828.95,E2 -14828.95} C_VEL
LIN {X 0,Y 326.546,Z 315.998,A -85,B 0,C 180,E1 -14833.071,E2 -14833.071} C_VEL
LIN {X 0,Y 327.621,Z 331.643,A -85,B 0,C 180,E1 -14833.63,E2 -14833.63} C_VEL
LIN {X 0,Y 329.103,Z 347.672,A -85,B 0,C 180,E1 -14834.175,E2 -14834.175} C_VEL
LIN {X 0,Y 328.138,Z 395.261,A -85,B 0,C 180,E1 -14835.704,E2 -14835.704} C_VEL
LIN {X 0,Y 327.705,Z 407.686,A -85,B 0,C 180,E1 -14836.357,E2 -14836.357} C_VEL
LIN {X 0,Y 327.175,Z 417.923,A -85,B 0,C 180,E1 -14837.125,E2 -14837.125} C_VEL
LIN {X 0,Y 326.627,Z 427.51,A -85,B 0,C 180,E1 -14838.05,E2 -14838.05} C_VEL
LIN {X 0,Y 326.191,Z 437.624,A -85,B 0,C 180,E1 -14839.293,E2 -14839.293} C_VEL
LIN {X 0,Y 325.72,Z 446.431,A -85,B 0,C 180,E1 -14840.689,E2 -14840.689} C_VEL
LIN {X 0,Y 325.47,Z 452.855,A -85,B 0,C 180,E1 -14841.934,E2 -14841.934} C_VEL
LIN {X 0,Y 325.291,Z 458.171,A -85,B 0,C 180,E1 -14843.178,E2 -14843.178} C_VEL
LIN {X 0,Y 325.147,Z 463.423,A -85,B 0,C 180,E1 -14844.688,E2 -14844.688} C_VEL
LIN {X 0,Y 325.001,Z 467.743,A -85,B 0,C 180,E1 -14846.283,E2 -14846.283} C_VEL
LIN {X 0,Y 324.967,Z 470.246,A -85,B 0,C 180,E1 -14847.523,E2 -14847.523} C_VEL
LIN {X 0,Y 325.084,Z 472.158,A -85,B 0,C 180,E1 -14848.763,E2 -14848.763} C_VEL
LIN {X 0,Y 325.153,Z 473.501,A -85,B 0,C 180,E1 -14850.002,E2 -14850.002} C_VEL
LIN {X 0,Y 324.877,Z 474.292,A -85,B 0,C 180,E1 -14851.242,E2 -14851.242} C_VEL
LIN {X 0,Y 324.856,Z 474.523,A -85,B 0,C 180,E1 -14852.482,E2 -14852.482} C_VEL
LIN {X 0,Y 324.934,Z 474.138,A -85,B 0,C 180,E1 -14853.722,E2 -14853.722} C_VEL
LIN {X 0,Y 325.083,Z 472.13,A -85,B 0,C 180,E1 -14855.995,E2 -14855.995} C_VEL
LIN {X 0,Y 325.587,Z 468.614,A -85,B 0,C 180,E1 -14858.068,E2 -14858.068} C_VEL
LIN {X 0,Y 326.071,Z 465.749,A -85,B 0,C 180,E1 -14859.305,E2 -14859.305} C_VEL
LIN {X 0,Y 327.098,Z 460.199,A -85,B 0,C 180,E1 -14861.152,E2 -14861.152} C_VEL
LIN {X 0,Y 328.452,Z 452.928,A -85,B 0,C 180,E1 -14862.986,E2 -14862.986} C_VEL
LIN {X 0,Y 329.759,Z 445.134,A -85,B 0,C 180,E1 -14864.504,E2 -14864.504} C_VEL
LIN {X 0,Y 330.881,Z 438.632,A -85,B 0,C 180,E1 -14865.557,E2 -14865.557} C_VEL
LIN {X 0,Y 332.202,Z 430.874,A -85,B 0,C 180,E1 -14866.597,E2 -14866.597} C_VEL
LIN {X 0,Y 333.669,Z 421.437,A -85,B 0,C 180,E1 -14867.626,E2 -14867.626} C_VEL
LIN {X 0,Y 335.293,Z 410.123,A -85,B 0,C 180,E1 -14868.565,E2 -14868.565} C_VEL
LIN {X 0,Y 336.491,Z 399.66,A -85,B 0,C 180,E1 -14869.207,E2 -14869.207} C_VEL
LIN {X 0,Y 337.551,Z 387.394,A -85,B 0,C 180,E1 -14869.75,E2 -14869.75} C_VEL
LIN {X 0,Y 339.814,Z 349.659,A -85,B 0,C 180,E1 -14871.082,E2 -14871.082} C_VEL
LIN {X 0,Y 338.221,Z 337.264,A -85,B 0,C 180,E1 -14871.828,E2 -14871.828} C_VEL
LIN {X 0,Y 335.436,Z 323.137,A -85,B 0,C 180,E1 -14872.873,E2 -14872.873} C_VEL
LIN {X 0,Y 332.083,Z 309.999,A -85,B 0,C 180,E1 -14874.031,E2 -14874.031} C_VEL
LIN {X 0,Y 332.434,Z 306.308,A -85,B 0,C 180,E1 -14875.015,E2 -14875.015} C_VEL
LIN {X 0,Y 330.54,Z 297.443,A -85,B 0,C 180,E1 -14877.891,E2 -14877.891} C_VEL
LIN {X 0,Y 328.457,Z 290.268,A -85,B 0,C 180,E1 -14880.531,E2 -14880.531} C_VEL
LIN {X 0,Y 326.593,Z 284.616,A -85,B 0,C 180,E1 -14882.933,E2 -14882.933} C_VEL
LIN {X 0,Y 326.632,Z 284.611,A -85,B 0,C 180,E1 -14887.049,E2 -14887.049} C_VEL
LIN {X 0,Y 326.568,Z 284.616,A -85,B 0,C 180,E1 -14890.214,E2 -14890.214} C_VEL
LIN {X 0,Y 326.542,Z 284.619,A -85,B 0,C 180,E1 -14893.531,E2 -14893.531} C_VEL
LIN {X 0,Y 326.551,Z 284.621,A -85,B 0,C 180,E1 -14897.035,E2 -14897.035} C_VEL
LIN {X 0,Y 326.606,Z 284.612,A -85,B 0,C 180,E1 -14900.776,E2 -14900.776} C_VEL
LIN {X 0,Y 326.63,Z 284.609,A -85,B 0,C 180,E1 -14904.477,E2 -14904.477} C_VEL
LIN {X 0,Y 326.627,Z 284.609,A -85,B 0,C 180,E1 -14907.452,E2 -14907.452} C_VEL
LIN {X 0,Y 326.635,Z 284.612,A -85,B 0,C 180,E1 -14910.333,E2 -14910.333} C_VEL
LIN {X 0,Y 326.667,Z 284.72,A -85,B 0,C 180,E1 -14912.529,E2 -14912.529} C_VEL
LIN {X 0,Y 329.757,Z 293.117,A -85,B 0,C 180,E1 -14915.549,E2 -14915.549} C_VEL
LIN {X 0,Y 335.254,Z 302.544,A -85,B 0,C 180,E1 -14916.931,E2 -14916.931} C_VEL
LIN {X 0,Y 339.933,Z 311.82,A -85,B 0,C 180,E1 -14918.061,E2 -14918.061} C_VEL
LIN {X 0,Y 341.352,Z 315.201,A -85,B 0,C 180,E1 -14918.412,E2 -14918.412} C_VEL
LIN {X 0,Y 341.509,Z 318.295,A -85,B 0,C 180,E1 -14918.571,E2 -14918.571} C_VEL
LIN {X 0,Y 337.741,Z 374.428,A -85,B 0,C 180,E1 -14920.587,E2 -14920.587} C_VEL
LIN {X 0,Y 336.639,Z 386.528,A -85,B 0,C 180,E1 -14921.272,E2 -14921.272} C_VEL
LIN {X 0,Y 335.61,Z 396.023,A -85,B 0,C 180,E1 -14922.003,E2 -14922.003} C_VEL
LIN {X 0,Y 334.415,Z 405.1,A -85,B 0,C 180,E1 -14922.884,E2 -14922.884} C_VEL
LIN {X 0,Y 332.987,Z 414.789,A -85,B 0,C 180,E1 -14924.07,E2 -14924.07} C_VEL
LIN {X 0,Y 331.729,Z 422.447,A -85,B 0,C 180,E1 -14925.267,E2 -14925.267} C_VEL
LIN {X 0,Y 330.582,Z 428.8,A -85,B 0,C 180,E1 -14926.47,E2 -14926.47} C_VEL
LIN {X 0,Y 329.22,Z 435.33,A -85,B 0,C 180,E1 -14927.981,E2 -14927.981} C_VEL
LIN {X 0,Y 328.055,Z 440.582,A -85,B 0,C 180,E1 -14929.502,E2 -14929.502} C_VEL
LIN {X 0,Y 327.149,Z 445.398,A -85,B 0,C 180,E1 -14931.345,E2 -14931.345} C_VEL
LIN {X 0,Y 326.419,Z 447.755,A -85,B 0,C 180,E1 -14932.572,E2 -14932.572} C_VEL
LIN {X 0,Y 325.86,Z 449.518,A -85,B 0,C 180,E1 -14933.803,E2 -14933.803} C_VEL
LIN {X 0,Y 325.648,Z 450.732,A -85,B 0,C 180,E1 -14935.042,E2 -14935.042} C_VEL
LIN {X 0,Y 325.392,Z 451.458,A -85,B 0,C 180,E1 -14936.279,E2 -14936.279} C_VEL
LIN {X 0,Y 325.141,Z 451.66,A -85,B 0,C 180,E1 -14937.516,E2 -14937.516} C_VEL
LIN {X 0,Y 324.978,Z 451.237,A -85,B 0,C 180,E1 -14938.755,E2 -14938.755} C_VEL
LIN {X 0,Y 324.923,Z 450.264,A -85,B 0,C 180,E1 -14939.994,E2 -14939.994} C_VEL
LIN {X 0,Y 324.899,Z 447.858,A -85,B 0,C 180,E1 -14941.853,E2 -14941.853} C_VEL
LIN {X 0,Y 325.101,Z 444.08,A -85,B 0,C 180,E1 -14943.712,E2 -14943.712} C_VEL
LIN {X 0,Y 325.172,Z 439.357,A -85,B 0,C 180,E1 -14945.384,E2 -14945.384} C_VEL
LIN {X 0,Y 325.41,Z 434.502,A -85,B 0,C 180,E1 -14946.753,E2 -14946.753} C_VEL
LIN {X 0,Y 325.701,Z 428.869,A -85,B 0,C 180,E1 -14948.056,E2 -14948.056} C_VEL
LIN {X 0,Y 326.016,Z 422.358,A -85,B 0,C 180,E1 -14949.298,E2 -14949.298} C_VEL
LIN {X 0,Y 326.359,Z 414.468,A -85,B 0,C 180,E1 -14950.54,E2 -14950.54} C_VEL
LIN {X 0,Y 326.96,Z 404.739,A -85,B 0,C 180,E1 -14951.776,E2 -14951.776} C_VEL
LIN {X 0,Y 327.318,Z 395.313,A -85,B 0,C 180,E1 -14952.707,E2 -14952.707} C_VEL
LIN {X 0,Y 327.715,Z 386.497,A -85,B 0,C 180,E1 -14953.401,E2 -14953.401} C_VEL
LIN {X 0,Y 328.101,Z 376.276,A -85,B 0,C 180,E1 -14954.016,E2 -14954.016} C_VEL
LIN {X 0,Y 328.313,Z 364.127,A -85,B 0,C 180,E1 -14954.521,E2 -14954.521} C_VEL
LIN {X 0,Y 329.366,Z 311.91,A -85,B 0,C 180,E1 -14956.152,E2 -14956.152} C_VEL
LIN {X 0,Y 326.829,Z 291.899,A -85,B 0,C 180,E1 -14956.868,E2 -14956.868} C_VEL
LIN {X 0,Y 326.925,Z 285.719,A -85,B 0,C 180,E1 -14958.932,E2 -14958.932} C_VEL
LIN {X 0,Y 326.813,Z 284.586,A -85,B 0,C 180,E1 -14959.372,E2 -14959.372} C_VEL
LIN {X 0,Y 326.599,Z 284.617,A -85,B 0,C 180,E1 -14964.125,E2 -14964.125} C_VEL
LIN {X 0,Y 326.574,Z 284.62,A -85,B 0,C 180,E1 -14968.25,E2 -14968.25} C_VEL
LIN {X 0,Y 326.553,Z 284.617,A -85,B 0,C 180,E1 -14971.09,E2 -14971.09} C_VEL
LIN {X 0,Y 326.587,Z 284.615,A -85,B 0,C 180,E1 -14974.012,E2 -14974.012} C_VEL
LIN {X 0,Y 326.6,Z 284.612,A -85,B 0,C 180,E1 -14977.23,E2 -14977.23} C_VEL
LIN {X 0,Y 326.518,Z 284.623,A -85,B 0,C 180,E1 -14981.117,E2 -14981.117} C_VEL
LIN {X 0,Y 326.532,Z 284.62,A -85,B 0,C 180,E1 -14983.519,E2 -14983.519} C_VEL
LIN {X 0,Y 326.544,Z 284.622,A -85,B 0,C 180,E1 -14987.021,E2 -14987.021} C_VEL
LIN {X 0,Y 326.577,Z 284.619,A -85,B 0,C 180,E1 -14990.767,E2 -14990.767} C_VEL
LIN {X 0,Y 326.575,Z 284.616,A -85,B 0,C 180,E1 -14994.474,E2 -14994.474} C_VEL
LIN {X 0,Y 326.569,Z 284.618,A -85,B 0,C 180,E1 -14997.449,E2 -14997.449} C_VEL
LIN {X 0,Y 326.592,Z 284.612,A -85,B 0,C 180,E1 -15000.332,E2 -15000.332} C_VEL
LIN {X 0,Y 326.635,Z 284.612,A -85,B 0,C 180,E1 -15003.136,E2 -15003.136} C_VEL
LIN {X 0,Y 326.606,Z 284.612,A -85,B 0,C 180,E1 -15005.866,E2 -15005.866} C_VEL
LIN {X 0,Y 326.608,Z 284.612,A -85,B 0,C 180,E1 -15009.86,E2 -15009.86} C_VEL
LIN {X 0,Y 326.649,Z 284.605,A -85,B 0,C 180,E1 -15012.467,E2 -15012.467} C_VEL
LIN {X 0,Y 326.71,Z 284.598,A -85,B 0,C 180,E1 -15016.311,E2 -15016.311} C_VEL
LIN {X 0,Y 326.763,Z 284.594,A -85,B 0,C 180,E1 -15020.09,E2 -15020.09} C_VEL
LIN {X 0,Y 326.94,Z 284.575,A -85,B 0,C 180,E1 -15023.828,E2 -15023.828} C_VEL
LIN {X 0,Y 327.023,Z 284.561,A -85,B 0,C 180,E1 -15027.535,E2 -15027.535} C_VEL
LIN {X 0,Y 327.164,Z 284.547,A -85,B 0,C 180,E1 -15029.998,E2 -15029.998} C_VEL
LIN {X 0,Y 327.022,Z 284.561,A -85,B 0,C 180,E1 -15032.461,E2 -15032.461} C_VEL
LIN {X 0,Y 326.936,Z 284.576,A -85,B 0,C 180,E1 -15036.168,E2 -15036.168} C_VEL
LIN {X 0,Y 326.759,Z 284.594,A -85,B 0,C 180,E1 -15039.906,E2 -15039.906} C_VEL
LIN {X 0,Y 326.705,Z 284.599,A -85,B 0,C 180,E1 -15043.685,E2 -15043.685} C_VEL
LIN {X 0,Y 326.642,Z 284.606,A -85,B 0,C 180,E1 -15047.529,E2 -15047.529} C_VEL
LIN {X 0,Y 326.6,Z 284.613,A -85,B 0,C 180,E1 -15050.136,E2 -15050.136} C_VEL
LIN {X 0,Y 326.596,Z 284.613,A -85,B 0,C 180,E1 -15054.131,E2 -15054.131} C_VEL
LIN {X 0,Y 326.632,Z 284.612,A -85,B 0,C 180,E1 -15056.86,E2 -15056.86} C_VEL
LIN {X 0,Y 326.587,Z 284.617,A -85,B 0,C 180,E1 -15060.613,E2 -15060.613} C_VEL
LIN {X 0,Y 326.556,Z 284.617,A -85,B 0,C 180,E1 -15064.022,E2 -15064.022} C_VEL
LIN {X 0,Y 326.579,Z 284.618,A -85,B 0,C 180,E1 -15067.242,E2 -15067.242} C_VEL
LIN {X 0,Y 326.587,Z 284.613,A -85,B 0,C 180,E1 -15070.206,E2 -15070.206} C_VEL
LIN {X 0,Y 326.611,Z 284.613,A -85,B 0,C 180,E1 -15073.514,E2 -15073.514} C_VEL
LIN {X 0,Y 326.606,Z 284.614,A -85,B 0,C 180,E1 -15077.019,E2 -15077.019} C_VEL
LIN {X 0,Y 326.601,Z 284.612,A -85,B 0,C 180,E1 -15080.771,E2 -15080.771} C_VEL
LIN {X 0,Y 326.572,Z 284.615,A -85,B 0,C 180,E1 -15084.485,E2 -15084.485} C_VEL
LIN {X 0,Y 326.569,Z 284.62,A -85,B 0,C 180,E1 -15087.461,E2 -15087.461} C_VEL
LIN {X 0,Y 326.611,Z 284.61,A -85,B 0,C 180,E1 -15090.345,E2 -15090.345} C_VEL
LIN {X 0,Y 326.616,Z 284.609,A -85,B 0,C 180,E1 -15092.564,E2 -15092.564} C_VEL
LIN {X 0,Y 325.969,Z 284.694,A -85,B 0,C 180,E1 -15093.592,E2 -15093.592} C_VEL
LIN {X 0,Y 323.106,Z 285.048,A -85,B 0,C 180,E1 -15095.265,E2 -15095.265} C_VEL
LIN {X 0,Y 320.666,Z 285.351,A -85,B 0,C 180,E1 -15096.621,E2 -15096.621} C_VEL
LIN {X 0,Y 319.62,Z 285.484,A -85,B 0,C 180,E1 -15097.67,E2 -15097.67} C_VEL
LIN {X 0,Y 319.537,Z 285.495,A -85,B 0,C 180,E1 -15098.026,E2 -15098.026} C_VEL
LIN {X 0,Y 319.585,Z 285.49,A -85,B 0,C 180,E1 -15102.077,E2 -15102.077} C_VEL
LIN {X 0,Y 319.705,Z 285.475,A -85,B 0,C 180,E1 -15106.014,E2 -15106.014} C_VEL
LIN {X 0,Y 319.712,Z 285.472,A -85,B 0,C 180,E1 -15109.878,E2 -15109.878} C_VEL
LIN {X 0,Y 319.897,Z 285.447,A -85,B 0,C 180,E1 -15113.7,E2 -15113.7} C_VEL
LIN {X 0,Y 320,Z 285.437,A -85,B 0,C 180,E1 -15118.748,E2 -15118.748} C_VEL
LIN {X 0,Y 319.962,Z 285.444,A -85,B 0,C 180,E1 -15122.524,E2 -15122.524} C_VEL
LIN {X 0,Y 319.888,Z 285.45,A -85,B 0,C 180,E1 -15126.313,E2 -15126.313} C_VEL
LIN {X 0,Y 319.724,Z 285.468,A -85,B 0,C 180,E1 -15130.134,E2 -15130.134} C_VEL
LIN {X 0,Y 319.701,Z 285.47,A -85,B 0,C 180,E1 -15133.999,E2 -15133.999} C_VEL
LIN {X 0,Y 319.58,Z 285.486,A -85,B 0,C 180,E1 -15137.937,E2 -15137.937} C_VEL
LIN {X 0,Y 319.558,Z 285.488,A -85,B 0,C 180,E1 -15141.961,E2 -15141.961} C_VEL
LIN {X 0,Y 319.549,Z 285.489,A -85,B 0,C 180,E1 -15146.101,E2 -15146.101} C_VEL
LIN {X 0,Y 319.541,Z 285.493,A -85,B 0,C 180,E1 -15148.944,E2 -15148.944} C_VEL
LIN {X 0,Y 319.523,Z 285.494,A -85,B 0,C 180,E1 -15151.868,E2 -15151.868} C_VEL
LIN {X 0,Y 319.578,Z 285.491,A -85,B 0,C 180,E1 -15155.547,E2 -15155.547} C_VEL
LIN {X 0,Y 319.531,Z 285.497,A -85,B 0,C 180,E1 -15159.667,E2 -15159.667} C_VEL
LIN {X 0,Y 319.52,Z 285.497,A -85,B 0,C 180,E1 -15163.464,E2 -15163.464} C_VEL
LIN {X 0,Y 319.553,Z 285.489,A -85,B 0,C 180,E1 -15167.02,E2 -15167.02} C_VEL
LIN {X 0,Y 319.521,Z 285.495,A -85,B 0,C 180,E1 -15170.37,E2 -15170.37} C_VEL
LIN {X 0,Y 319.584,Z 285.487,A -85,B 0,C 180,E1 -15174.462,E2 -15174.462} C_VEL
LIN {X 0,Y 319.529,Z 285.498,A -85,B 0,C 180,E1 -15178.141,E2 -15178.141} C_VEL
LIN {X 0,Y 319.552,Z 285.49,A -85,B 0,C 180,E1 -15181.617,E2 -15181.617} C_VEL
LIN {X 0,Y 319.684,Z 285.565,A -85,B 0,C 180,E1 -15183.7,E2 -15183.7} C_VEL
LIN {X 0,Y 321.228,Z 294.472,A -85,B 0,C 180,E1 -15186.504,E2 -15186.504} C_VEL
LIN {X 0,Y 320.594,Z 303.186,A -85,B 0,C 180,E1 -15189.134,E2 -15189.134} C_VEL
LIN {X 0,Y 319.495,Z 315.862,A -85,B 0,C 180,E1 -15192.933,E2 -15192.933} C_VEL
LIN {X 0,Y 320.529,Z 331.619,A -85,B 0,C 180,E1 -15193.496,E2 -15193.496} C_VEL
LIN {X 0,Y 322.041,Z 347.405,A -85,B 0,C 180,E1 -15194.047,E2 -15194.047} C_VEL
LIN {X 0,Y 321.064,Z 395.006,A -85,B 0,C 180,E1 -15195.625,E2 -15195.625} C_VEL
LIN {X 0,Y 320.625,Z 407.404,A -85,B 0,C 180,E1 -15196.292,E2 -15196.292} C_VEL
LIN {X 0,Y 320.135,Z 416.729,A -85,B 0,C 180,E1 -15196.998,E2 -15196.998} C_VEL
LIN {X 0,Y 319.68,Z 425.01,A -85,B 0,C 180,E1 -15197.786,E2 -15197.786} C_VEL
LIN {X 0,Y 319.239,Z 433.136,A -85,B 0,C 180,E1 -15198.735,E2 -15198.735} C_VEL
LIN {X 0,Y 318.88,Z 440.939,A -85,B 0,C 180,E1 -15199.847,E2 -15199.847} C_VEL
LIN {X 0,Y 318.487,Z 449.952,A -85,B 0,C 180,E1 -15201.436,E2 -15201.436} C_VEL
LIN {X 0,Y 318.241,Z 456.915,A -85,B 0,C 180,E1 -15203.026,E2 -15203.026} C_VEL
LIN {X 0,Y 318.093,Z 461.593,A -85,B 0,C 180,E1 -15204.336,E2 -15204.336} C_VEL
LIN {X 0,Y 318.036,Z 465.228,A -85,B 0,C 180,E1 -15205.566,E2 -15205.566} C_VEL
LIN {X 0,Y 317.886,Z 468.266,A -85,B 0,C 180,E1 -15206.834,E2 -15206.834} C_VEL
LIN {X 0,Y 318.013,Z 471.52,A -85,B 0,C 180,E1 -15208.736,E2 -15208.736} C_VEL
LIN {X 0,Y 318.092,Z 473.006,A -85,B 0,C 180,E1 -15210.002,E2 -15210.002} C_VEL
LIN {X 0,Y 317.787,Z 473.895,A -85,B 0,C 180,E1 -15211.269,E2 -15211.269} C_VEL
LIN {X 0,Y 317.778,Z 474.172,A -85,B 0,C 180,E1 -15212.537,E2 -15212.537} C_VEL
LIN {X 0,Y 317.845,Z 473.91,A -85,B 0,C 180,E1 -15213.806,E2 -15213.806} C_VEL
LIN {X 0,Y 318.003,Z 472.337,A -85,B 0,C 180,E1 -15215.971,E2 -15215.971} C_VEL
LIN {X 0,Y 318.356,Z 470.042,A -85,B 0,C 180,E1 -15217.614,E2 -15217.614} C_VEL
LIN {X 0,Y 319.07,Z 466.118,A -85,B 0,C 180,E1 -15219.511,E2 -15219.511} C_VEL
LIN {X 0,Y 319.956,Z 461.744,A -85,B 0,C 180,E1 -15221.083,E2 -15221.083} C_VEL
LIN {X 0,Y 321.111,Z 456.259,A -85,B 0,C 180,E1 -15222.644,E2 -15222.644} C_VEL
LIN {X 0,Y 322.391,Z 449.513,A -85,B 0,C 180,E1 -15224.198,E2 -15224.198} C_VEL
LIN {X 0,Y 323.979,Z 441.162,A -85,B 0,C 180,E1 -15225.735,E2 -15225.735} C_VEL
LIN {X 0,Y 325.751,Z 431.515,A -85,B 0,C 180,E1 -15227.097,E2 -15227.097} C_VEL
LIN {X 0,Y 327.294,Z 422.286,A -85,B 0,C 180,E1 -15228.143,E2 -15228.143} C_VEL
LIN {X 0,Y 329.159,Z 410.657,A -85,B 0,C 180,E1 -15229.166,E2 -15229.166} C_VEL
LIN {X 0,Y 330.417,Z 400.638,A -85,B 0,C 180,E1 -15229.817,E2 -15229.817} C_VEL
LIN {X 0,Y 331.506,Z 389.608,A -85,B 0,C 180,E1 -15230.341,E2 -15230.341} C_VEL
LIN {X 0,Y 334.033,Z 350.858,A -85,B 0,C 180,E1 -15231.757,E2 -15231.757} C_VEL
LIN {X 0,Y 332.442,Z 337.871,A -85,B 0,C 180,E1 -15232.594,E2 -15232.594} C_VEL
LIN {X 0,Y 329.509,Z 323.379,A -85,B 0,C 180,E1 -15233.742,E2 -15233.742} C_VEL
LIN {X 0,Y 326.535,Z 311.898,A -85,B 0,C 180,E1 -15234.839,E2 -15234.839} C_VEL
LIN {X 0,Y 325.91,Z 309.355,A -85,B 0,C 180,E1 -15235.115,E2 -15235.115} C_VEL
LIN {X 0,Y 324.916,Z 303.522,A -85,B 0,C 180,E1 -15237.018,E2 -15237.018} C_VEL
LIN {X 0,Y 323.177,Z 296.526,A -85,B 0,C 180,E1 -15239.55,E2 -15239.55} C_VEL
LIN {X 0,Y 320.883,Z 289.55,A -85,B 0,C 180,E1 -15242.454,E2 -15242.454} C_VEL
LIN {X 0,Y 319.532,Z 285.495,A -85,B 0,C 180,E1 -15244.403,E2 -15244.403} C_VEL
LIN {X 0,Y 319.536,Z 285.492,A -85,B 0,C 180,E1 -15248.015,E2 -15248.015} C_VEL
LIN {X 0,Y 319.51,Z 285.495,A -85,B 0,C 180,E1 -15251.588,E2 -15251.588} C_VEL
LIN {X 0,Y 319.496,Z 285.498,A -85,B 0,C 180,E1 -15255.253,E2 -15255.253} C_VEL
LIN {X 0,Y 319.507,Z 285.497,A -85,B 0,C 180,E1 -15258.703,E2 -15258.703} C_VEL
LIN {X 0,Y 319.56,Z 285.487,A -85,B 0,C 180,E1 -15262.351,E2 -15262.351} C_VEL
LIN {X 0,Y 319.578,Z 285.487,A -85,B 0,C 180,E1 -15265.12,E2 -15265.12} C_VEL
LIN {X 0,Y 319.543,Z 285.495,A -85,B 0,C 180,E1 -15268.134,E2 -15268.134} C_VEL
LIN {X 0,Y 319.587,Z 285.685,A -85,B 0,C 180,E1 -15270.971,E2 -15270.971} C_VEL
LIN {X 0,Y 322.631,Z 293.639,A -85,B 0,C 180,E1 -15274.25,E2 -15274.25} C_VEL
LIN {X 0,Y 326.692,Z 300.269,A -85,B 0,C 180,E1 -15275.395,E2 -15275.395} C_VEL
LIN {X 0,Y 331.457,Z 308.634,A -85,B 0,C 180,E1 -15276.65,E2 -15276.65} C_VEL
LIN {X 0,Y 335.917,Z 317.94,A -85,B 0,C 180,E1 -15277.778,E2 -15277.778} C_VEL
LIN {X 0,Y 333.176,Z 356.763,A -85,B 0,C 180,E1 -15279.223,E2 -15279.223} C_VEL
LIN {X 0,Y 331.757,Z 376.463,A -85,B 0,C 180,E1 -15279.98,E2 -15279.98} C_VEL
LIN {X 0,Y 330.605,Z 387.915,A -85,B 0,C 180,E1 -15280.676,E2 -15280.676} C_VEL
LIN {X 0,Y 329.378,Z 397.924,A -85,B 0,C 180,E1 -15281.489,E2 -15281.489} C_VEL
LIN {X 0,Y 327.936,Z 407.947,A -85,B 0,C 180,E1 -15282.535,E2 -15282.535} C_VEL
LIN {X 0,Y 326.384,Z 416.92,A -85,B 0,C 180,E1 -15283.739,E2 -15283.739} C_VEL
LIN {X 0,Y 325.068,Z 424.297,A -85,B 0,C 180,E1 -15284.958,E2 -15284.958} C_VEL
LIN {X 0,Y 323.833,Z 430.428,A -85,B 0,C 180,E1 -15286.183,E2 -15286.183} C_VEL
LIN {X 0,Y 322.673,Z 435.556,A -85,B 0,C 180,E1 -15287.414,E2 -15287.414} C_VEL
LIN {X 0,Y 321.655,Z 439.83,A -85,B 0,C 180,E1 -15288.653,E2 -15288.653} C_VEL
LIN {X 0,Y 320.808,Z 443.362,A -85,B 0,C 180,E1 -15289.901,E2 -15289.901} C_VEL
LIN {X 0,Y 320.203,Z 446.255,A -85,B 0,C 180,E1 -15291.156,E2 -15291.156} C_VEL
LIN {X 0,Y 319.432,Z 448.553,A -85,B 0,C 180,E1 -15292.408,E2 -15292.408} C_VEL
LIN {X 0,Y 318.843,Z 450.193,A -85,B 0,C 180,E1 -15293.666,E2 -15293.666} C_VEL
LIN {X 0,Y 318.586,Z 451.259,A -85,B 0,C 180,E1 -15294.932,E2 -15294.932} C_VEL
LIN {X 0,Y 318.317,Z 451.831,A -85,B 0,C 180,E1 -15296.196,E2 -15296.196} C_VEL
LIN {X 0,Y 318.057,Z 451.905,A -85,B 0,C 180,E1 -15297.461,E2 -15297.461} C_VEL
LIN {X 0,Y 317.886,Z 451.435,A -85,B 0,C 180,E1 -15298.727,E2 -15298.727} C_VEL
LIN {X 0,Y 317.829,Z 450.343,A -85,B 0,C 180,E1 -15299.994,E2 -15299.994} C_VEL
LIN {X 0,Y 317.814,Z 447.751,A -85,B 0,C 180,E1 -15301.894,E2 -15301.894} C_VEL
LIN {X 0,Y 318.033,Z 443.707,A -85,B 0,C 180,E1 -15303.795,E2 -15303.795} C_VEL
LIN {X 0,Y 318.093,Z 438.023,A -85,B 0,C 180,E1 -15305.744,E2 -15305.744} C_VEL
LIN {X 0,Y 318.515,Z 430.888,A -85,B 0,C 180,E1 -15307.601,E2 -15307.601} C_VEL
LIN {X 0,Y 318.785,Z 424.719,A -85,B 0,C 180,E1 -15308.871,E2 -15308.871} C_VEL
LIN {X 0,Y 319.198,Z 417.257,A -85,B 0,C 180,E1 -15310.138,E2 -15310.138} C_VEL
LIN {X 0,Y 319.574,Z 409.35,A -85,B 0,C 180,E1 -15311.248,E2 -15311.248} C_VEL
LIN {X 0,Y 319.939,Z 402.643,A -85,B 0,C 180,E1 -15312.038,E2 -15312.038} C_VEL
LIN {X 0,Y 320.26,Z 394.576,A -85,B 0,C 180,E1 -15312.83,E2 -15312.83} C_VEL
LIN {X 0,Y 320.735,Z 384.485,A -85,B 0,C 180,E1 -15313.617,E2 -15313.617} C_VEL
LIN {X 0,Y 321.077,Z 372.76,A -85,B 0,C 180,E1 -15314.289,E2 -15314.289} C_VEL
LIN {X 0,Y 321.632,Z 349.808,A -85,B 0,C 180,E1 -15315.072,E2 -15315.072} C_VEL
LIN {X 0,Y 322.288,Z 312.361,A -85,B 0,C 180,E1 -15316.284,E2 -15316.284} C_VEL
LIN {X 0,Y 319.789,Z 292.353,A -85,B 0,C 180,E1 -15317.004,E2 -15317.004} C_VEL
LIN {X 0,Y 319.829,Z 286.044,A -85,B 0,C 180,E1 -15319.106,E2 -15319.106} C_VEL
LIN {X 0,Y 319.777,Z 285.463,A -85,B 0,C 180,E1 -15319.407,E2 -15319.407} C_VEL
LIN {X 0,Y 319.531,Z 285.492,A -85,B 0,C 180,E1 -15323.314,E2 -15323.314} C_VEL
LIN {X 0,Y 319.536,Z 285.496,A -85,B 0,C 180,E1 -15326.088,E2 -15326.088} C_VEL
LIN {X 0,Y 319.508,Z 285.495,A -85,B 0,C 180,E1 -15328.933,E2 -15328.933} C_VEL
LIN {X 0,Y 319.505,Z 285.496,A -85,B 0,C 180,E1 -15331.855,E2 -15331.855} C_VEL
LIN {X 0,Y 319.558,Z 285.488,A -85,B 0,C 180,E1 -15335.535,E2 -15335.535} C_VEL
LIN {X 0,Y 319.508,Z 285.496,A -85,B 0,C 180,E1 -15338.006,E2 -15338.006} C_VEL
LIN {X 0,Y 319.478,Z 285.498,A -85,B 0,C 180,E1 -15341.585,E2 -15341.585} C_VEL
LIN {X 0,Y 319.458,Z 285.507,A -85,B 0,C 180,E1 -15344.736,E2 -15344.736} C_VEL
LIN {X 0,Y 319.494,Z 285.498,A -85,B 0,C 180,E1 -15348.396,E2 -15348.396} C_VEL
LIN {X 0,Y 319.507,Z 285.495,A -85,B 0,C 180,E1 -15351.981,E2 -15351.981} C_VEL
LIN {X 0,Y 319.523,Z 285.498,A -85,B 0,C 180,E1 -15355.117,E2 -15355.117} C_VEL
LIN {X 0,Y 319.485,Z 285.497,A -85,B 0,C 180,E1 -15358.131,E2 -15358.131} C_VEL
LIN {X 0,Y 319.568,Z 285.49,A -85,B 0,C 180,E1 -15361.585,E2 -15361.585} C_VEL
LIN {X 0,Y 319.561,Z 285.494,A -85,B 0,C 180,E1 -15365.298,E2 -15365.298} C_VEL
LIN {X 0,Y 319.554,Z 285.495,A -85,B 0,C 180,E1 -15369.395,E2 -15369.395} C_VEL
LIN {X 0,Y 319.61,Z 285.483,A -85,B 0,C 180,E1 -15372.068,E2 -15372.068} C_VEL
LIN {X 0,Y 319.683,Z 285.475,A -85,B 0,C 180,E1 -15376.004,E2 -15376.004} C_VEL
LIN {X 0,Y 319.707,Z 285.474,A -85,B 0,C 180,E1 -15379.869,E2 -15379.869} C_VEL
LIN {X 0,Y 319.87,Z 285.45,A -85,B 0,C 180,E1 -15382.423,E2 -15382.423} C_VEL
LIN {X 0,Y 319.7,Z 285.471,A -85,B 0,C 180,E1 -15384.953,E2 -15384.953} C_VEL
LIN {X 0,Y 319.964,Z 285.44,A -85,B 0,C 180,E1 -15387.48,E2 -15387.48} C_VEL
LIN {X 0,Y 320.115,Z 285.425,A -85,B 0,C 180,E1 -15389.998,E2 -15389.998} C_VEL
LIN {X 0,Y 319.962,Z 285.44,A -85,B 0,C 180,E1 -15392.516,E2 -15392.516} C_VEL
LIN {X 0,Y 319.891,Z 285.452,A -85,B 0,C 180,E1 -15396.304,E2 -15396.304} C_VEL
LIN {X 0,Y 319.785,Z 285.461,A -85,B 0,C 180,E1 -15398.847,E2 -15398.847} C_VEL
LIN {X 0,Y 319.63,Z 285.482,A -85,B 0,C 180,E1 -15402.7,E2 -15402.7} C_VEL
LIN {X 0,Y 319.63,Z 285.479,A -85,B 0,C 180,E1 -15405.296,E2 -15405.296} C_VEL
LIN {X 0,Y 319.597,Z 285.484,A -85,B 0,C 180,E1 -15409.257,E2 -15409.257} C_VEL
LIN {X 0,Y 319.508,Z 285.495,A -85,B 0,C 180,E1 -15413.321,E2 -15413.321} C_VEL
LIN {X 0,Y 319.566,Z 285.488,A -85,B 0,C 180,E1 -15416.091,E2 -15416.091} C_VEL
LIN {X 0,Y 319.538,Z 285.496,A -85,B 0,C 180,E1 -15418.936,E2 -15418.936} C_VEL
LIN {X 0,Y 319.481,Z 285.498,A -85,B 0,C 180,E1 -15421.864,E2 -15421.864} C_VEL
LIN {X 0,Y 319.529,Z 285.493,A -85,B 0,C 180,E1 -15425.546,E2 -15425.546} C_VEL
LIN {X 0,Y 319.535,Z 285.491,A -85,B 0,C 180,E1 -15428.01,E2 -15428.01} C_VEL
LIN {X 0,Y 319.555,Z 285.491,A -85,B 0,C 180,E1 -15431.616,E2 -15431.616} C_VEL
LIN {X 0,Y 319.6,Z 285.489,A -85,B 0,C 180,E1 -15435.289,E2 -15435.289} C_VEL
LIN {X 0,Y 319.539,Z 285.491,A -85,B 0,C 180,E1 -15438.725,E2 -15438.725} C_VEL
LIN {X 0,Y 319.541,Z 285.491,A -85,B 0,C 180,E1 -15442.348,E2 -15442.348} C_VEL
LIN {X 0,Y 319.52,Z 285.495,A -85,B 0,C 180,E1 -15445.128,E2 -15445.128} C_VEL
LIN {X 0,Y 319.529,Z 285.493,A -85,B 0,C 180,E1 -15449.065,E2 -15449.065} C_VEL
LIN {X 0,Y 319.568,Z 285.487,A -85,B 0,C 180,E1 -15452.554,E2 -15452.554} C_VEL
LIN {X 0,Y 319.57,Z 285.488,A -85,B 0,C 180,E1 -15455.31,E2 -15455.31} C_VEL
LIN {X 0,Y 319.537,Z 285.495,A -85,B 0,C 180,E1 -15458.026,E2 -15458.026} C_VEL
LIN {X 0,Y 318.874,Z 285.582,A -85,B 0,C 180,E1 -15459.079,E2 -15459.079} C_VEL
LIN {X 0,Y 316.032,Z 285.934,A -85,B 0,C 180,E1 -15460.794,E2 -15460.794} C_VEL
LIN {X 0,Y 313.634,Z 286.231,A -85,B 0,C 180,E1 -15462.183,E2 -15462.183} C_VEL
LIN {X 0,Y 312.624,Z 286.352,A -85,B 0,C 180,E1 -15463.259,E2 -15463.259} C_VEL
LIN {X 0,Y 312.553,Z 286.36,A -85,B 0,C 180,E1 -15463.623,E2 -15463.623} C_VEL
LIN {X 0,Y 312.659,Z 286.35,A -85,B 0,C 180,E1 -15465.692,E2 -15465.692} C_VEL
LIN {X 0,Y 312.662,Z 286.349,A -85,B 0,C 180,E1 -15469.648,E2 -15469.648} C_VEL
